KUKA KRL program: test1.src, test1.dat

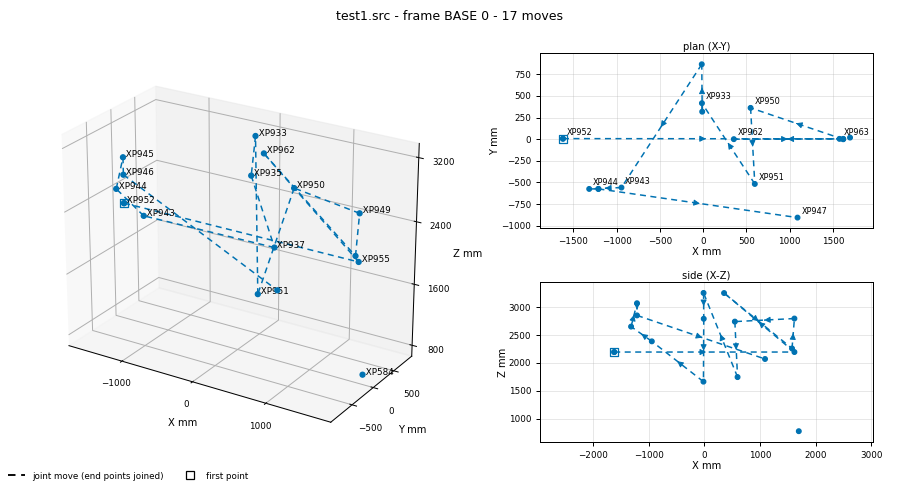
[picture p0: tool path of test1.src in frame BASE 0, 17 of 19 moves have a stored position in this frame; points joined in program order, loops and branches not executed]
--- test1.src ---
&ACCESS RVP
&REL 764
&PARAM TEMPLATE = C:\KRC\Roboter\Template\vorgabe
&PARAM EDITMASK = *
DEF test1( )
;FOLD INI;%{PE}%V3.2.0,%MKUKATPBASIS,%CINIT,%VCOMMON,%P
;FOLD BAS INI;%{E}%V3.2.0,%MKUKATPBASIS,%CINIT,%VINIT,%P
GLOBAL INTERRUPT DECL 3 WHEN $STOPMESS==TRUE DO IR_STOPM ( )
INTERRUPT ON 3
BAS (#INITMOV,0 )
;ENDFOLD (BAS INI)
;FOLD A20 INI;%{E}%V3.2.0,%MKUKATPA20,%CINIT,%VINIT,%P
IF ARC20==TRUE THEN
A20 (ARC_INI)
INTERRUPT DECL 6 WHEN $CYCFLAG[3]==FALSE DO A20(TECH_STOP2)
ENDIF
;ENDFOLD (A20 INI)
;FOLD A10 INI;%{E}%V3.2.0,%MKUKATPARC,%CINIT,%VINIT,%P
IF A10_OPTION==#ACTIVE THEN
INTERRUPT DECL 4 WHEN $CYCFLAG[2]==FALSE DO A10 (#APPL_ERROR)
INTERRUPT DECL 7 WHEN A_ARC_SWI==#ACTIVE DO A10 (#ARC_SEAM)
INTERRUPT DECL 5 WHEN A_FLY_ARC==TRUE DO A10 (#HPU_ARC)
INTERRUPT  ON 5
A10_INI ( )
ENDIF
;ENDFOLD (A10 INI)
;FOLD GRIPPER INI;%{E}%V3.2.0,%MKUKATPGRIPPER,%CINIT,%VINIT,%P
USER_GRP(0,DUMMY,DUMMY,GDEFAULT)
;ENDFOLD (GRIPPER INI)
;FOLD SPOT INI;%{E}%V3.2.0,%MKUKATPSPOT,%CINIT,%VINIT,%P
USERSPOT(#INIT)
;ENDFOLD (SPOT INI)
;FOLD TOUCHSENSE INI;%{E}%V3.2.0,%MKUKATPTS,%CINIT,%VINIT,%P
IF H70_OPTION THEN
INTERRUPT DECL 15 WHEN $MEAS_PULSE[TOUCH_I[TOUCH_ACTIVE].IN_NR] DO H70 (6,CD0 )
INTERRUPT DECL 16 WHEN $ZERO_MOVE DO H70 (7,CD0 )
INTERRUPT DECL 17 WHEN $TECHPAR_C[FG_TOUCH,8]>0.5 DO H70 (8,CD0)
H70 (1,CD0 )
ENDIF
;ENDFOLD (TOUCHSENSE INI)
;FOLD USER INI;%{E}%V3.2.0,%MKUKATPUSER,%CINIT,%VINIT,%P
;Make your modifications here
;ENDFOLD (USER INI)
;ENDFOLD (INI)
loop
;FOLD PTP HOME  Vel= 100 % DEFAULT;%{PE}%R 4.1.16,%MKUKATPBASIS,%CMOVE,%VPTP,%P 1:PTP, 2:HOME, 3:, 5:100, 7:DEFAULT
$BWDSTART = FALSE
PDAT_ACT=PDEFAULT
BAS(#PTP_DAT)
FDAT_ACT=FHOME
BAS(#FRAMES)
BAS(#VEL_PTP,100)
$H_POS=XHOME
PTP XHOME
;ENDFOLD


;FOLD WAIT Time= 2 sec;%{PE}%R 4.1.16,%MKUKATPBASIS,%CWAIT,%VWAIT,%P 2:2
WAIT SEC 2
;ENDFOLD

;FOLD PTP P952  Vel= 50 % PDAT628 Tool[1] Base[0];%{PE}%R 4.1.16,%MKUKATPBASIS,%CMOVE,%VPTP,%P 1:PTP, 2:P952, 3:, 5:50, 7:PDAT628
$BWDSTART = FALSE
PDAT_ACT=PPDAT628
BAS(#PTP_DAT)
FDAT_ACT=FP952
BAS(#FRAMES)
BAS(#VEL_PTP,50)
PTP XP952
;ENDFOLD
;FOLD PTP P954  Vel= 50 % PDAT630 Tool[1] Base[0];%{PE}%R 4.1.16,%MKUKATPBASIS,%CMOVE,%VPTP,%P 1:PTP, 2:P954, 3:, 5:50, 7:PDAT630
$BWDSTART = FALSE
PDAT_ACT=PPDAT630
BAS(#PTP_DAT)
FDAT_ACT=FP954
BAS(#FRAMES)
BAS(#VEL_PTP,50)
PTP XP954
;ENDFOLD
;FOLD PTP P955 CONT Vel= 100 % PDAT631 Tool[1]:Lexan Pointer Base[0];%{PE}%R 4.1.16,%MKUKATPBASIS,%CMOVE,%VPTP,%P 1:PTP, 2:P955, 3:C_PTP, 5:100, 7:PDAT631
$BWDSTART = FALSE
PDAT_ACT=PPDAT631
BAS(#PTP_DAT)
FDAT_ACT=FP955
BAS(#FRAMES)
BAS(#VEL_PTP,100)
PTP XP955 C_PTP
;ENDFOLD
;FOLD PTP P962 CONT Vel= 100 % PDAT638 Tool[1]:Lexan Pointer Base[0];%{PE}%R 4.1.16,%MKUKATPBASIS,%CMOVE,%VPTP,%P 1:PTP, 2:P962, 3:C_PTP, 5:100, 7:PDAT638
$BWDSTART = FALSE
PDAT_ACT=PPDAT638
BAS(#PTP_DAT)
FDAT_ACT=FP962
BAS(#FRAMES)
BAS(#VEL_PTP,100)
PTP XP962 C_PTP
;ENDFOLD
;FOLD PTP P963 CONT Vel= 100 % PDAT639 Tool[1]:Lexan Pointer Base[0];%{PE}%R 4.1.16,%MKUKATPBASIS,%CMOVE,%VPTP,%P 1:PTP, 2:P963, 3:C_PTP, 5:100, 7:PDAT639
$BWDSTART = FALSE
PDAT_ACT=PPDAT639
BAS(#PTP_DAT)
FDAT_ACT=FP963
BAS(#FRAMES)
BAS(#VEL_PTP,100)
PTP XP963 C_PTP
;ENDFOLD
;FOLD PTP P949 CONT Vel= 100 % PDAT625 Tool[1]:Lexan Pointer Base[0];%{PE}%R 4.1.16,%MKUKATPBASIS,%CMOVE,%VPTP,%P 1:PTP, 2:P949, 3:C_PTP, 5:100, 7:PDAT625
$BWDSTART = FALSE
PDAT_ACT=PPDAT625
BAS(#PTP_DAT)
FDAT_ACT=FP949
BAS(#FRAMES)
BAS(#VEL_PTP,100)
PTP XP949 C_PTP
;ENDFOLD

;FOLD PTP P950 CONT Vel= 100 % PDAT626 Tool[1]:Lexan Pointer Base[0];%{PE}%R 4.1.16,%MKUKATPBASIS,%CMOVE,%VPTP,%P 1:PTP, 2:P950, 3:C_PTP, 5:100, 7:PDAT626
$BWDSTART = FALSE
PDAT_ACT=PPDAT626
BAS(#PTP_DAT)
FDAT_ACT=FP950
BAS(#FRAMES)
BAS(#VEL_PTP,100)
PTP XP950 C_PTP
;ENDFOLD
;FOLD PTP P951 CONT Vel= 100 % PDAT627 Tool[1]:Lexan Pointer Base[0];%{PE}%R 4.1.16,%MKUKATPBASIS,%CMOVE,%VPTP,%P 1:PTP, 2:P951, 3:C_PTP, 5:100, 7:PDAT627
$BWDSTART = FALSE
PDAT_ACT=PPDAT627
BAS(#PTP_DAT)
FDAT_ACT=FP951
BAS(#FRAMES)
BAS(#VEL_PTP,100)
PTP XP951 C_PTP
;ENDFOLD
;FOLD PTP P933 CONT Vel= 100 % PDAT609 Tool[1]:Lexan Pointer Base[0];%{PE}%R 4.1.16,%MKUKATPBASIS,%CMOVE,%VPTP,%P 1:PTP, 2:P933, 3:C_PTP, 5:100, 7:PDAT609
$BWDSTART = FALSE
PDAT_ACT=PPDAT609
BAS(#PTP_DAT)
FDAT_ACT=FP933
BAS(#FRAMES)
BAS(#VEL_PTP,100)
PTP XP933 C_PTP
;ENDFOLD
;FOLD PTP P935 CONT Vel= 100 % PDAT611 Tool[1]:Lexan Pointer Base[0];%{PE}%R 4.1.16,%MKUKATPBASIS,%CMOVE,%VPTP,%P 1:PTP, 2:P935, 3:C_PTP, 5:100, 7:PDAT611
$BWDSTART = FALSE
PDAT_ACT=PPDAT611
BAS(#PTP_DAT)
FDAT_ACT=FP935
BAS(#FRAMES)
BAS(#VEL_PTP,100)
PTP XP935 C_PTP
;ENDFOLD
;FOLD PTP P937 CONT Vel= 100 % PDAT613 Tool[1]:Lexan Pointer Base[0];%{PE}%R 4.1.16,%MKUKATPBASIS,%CMOVE,%VPTP,%P 1:PTP, 2:P937, 3:C_PTP, 5:100, 7:PDAT613
$BWDSTART = FALSE
PDAT_ACT=PPDAT613
BAS(#PTP_DAT)
FDAT_ACT=FP937
BAS(#FRAMES)
BAS(#VEL_PTP,100)
PTP XP937 C_PTP
;ENDFOLD



;FOLD ; Robot is now at ship;%{PE}%R 4.1.16,%MKUKATPBASIS,%CCOMMENT,%VNORMAL,%P 2:Robot is now at ship
;ENDFOLD

;FOLD PTP P943 CONT Vel= 100 % PDAT619 Tool[1]:Lexan Pointer Base[0];%{PE}%R 4.1.16,%MKUKATPBASIS,%CMOVE,%VPTP,%P 1:PTP, 2:P943, 3:C_PTP, 5:100, 7:PDAT619
$BWDSTART = FALSE
PDAT_ACT=PPDAT619
BAS(#PTP_DAT)
FDAT_ACT=FP943
BAS(#FRAMES)
BAS(#VEL_PTP,100)
PTP XP943 C_PTP
;ENDFOLD
;FOLD PTP P944 CONT Vel= 100 % PDAT620 Tool[1]:Lexan Pointer Base[0];%{PE}%R 4.1.16,%MKUKATPBASIS,%CMOVE,%VPTP,%P 1:PTP, 2:P944, 3:C_PTP, 5:100, 7:PDAT620
$BWDSTART = FALSE
PDAT_ACT=PPDAT620
BAS(#PTP_DAT)
FDAT_ACT=FP944
BAS(#FRAMES)
BAS(#VEL_PTP,100)
PTP XP944 C_PTP
;ENDFOLD
;FOLD PTP P945 CONT Vel= 100 % PDAT621 Tool[1]:Lexan Pointer Base[0];%{PE}%R 4.1.16,%MKUKATPBASIS,%CMOVE,%VPTP,%P 1:PTP, 2:P945, 3:C_PTP, 5:100, 7:PDAT621
$BWDSTART = FALSE
PDAT_ACT=PPDAT621
BAS(#PTP_DAT)
FDAT_ACT=FP945
BAS(#FRAMES)
BAS(#VEL_PTP,100)
PTP XP945 C_PTP
;ENDFOLD
;FOLD PTP P946 CONT Vel= 100 % PDAT622 Tool[1]:Lexan Pointer Base[0];%{PE}%R 4.1.16,%MKUKATPBASIS,%CMOVE,%VPTP,%P 1:PTP, 2:P946, 3:C_PTP, 5:100, 7:PDAT622
$BWDSTART = FALSE
PDAT_ACT=PPDAT622
BAS(#PTP_DAT)
FDAT_ACT=FP946
BAS(#FRAMES)
BAS(#VEL_PTP,100)
PTP XP946 C_PTP
;ENDFOLD
;FOLD PTP P947 CONT Vel= 100 % PDAT623 Tool[1]:Lexan Pointer Base[0];%{PE}%R 4.1.16,%MKUKATPBASIS,%CMOVE,%VPTP,%P 1:PTP, 2:P947, 3:C_PTP, 5:100, 7:PDAT623
$BWDSTART = FALSE
PDAT_ACT=PPDAT623
BAS(#PTP_DAT)
FDAT_ACT=FP947
BAS(#FRAMES)
BAS(#VEL_PTP,100)
PTP XP947 C_PTP
;ENDFOLD

;FOLD ; Begin with tower 1;%{PE}%R 4.1.16,%MKUKATPBASIS,%CCOMMENT,%VNORMAL,%P 2:Begin with tower 1
;ENDFOLD


;FOLD ; tower 2 done;%{PE}%R 4.1.16,%MKUKATPBASIS,%CCOMMENT,%VNORMAL,%P 2:tower 2 done
;ENDFOLD
;FOLD ; approach;%{PE}%R 4.1.16,%MKUKATPBASIS,%CCOMMENT,%VNORMAL,%P 2:approach
;ENDFOLD



;FOLD ; foreword approach;%{PE}%R 4.1.16,%MKUKATPBASIS,%CCOMMENT,%VNORMAL,%P 2:foreword approach
;ENDFOLD







;FOLD ; mouth;%{PE}%R 4.1.16,%MKUKATPBASIS,%CCOMMENT,%VNORMAL,%P 2:mouth
;ENDFOLD

;FOLD ; top vert orbit;%{PE}%R 4.1.16,%MKUKATPBASIS,%CCOMMENT,%VNORMAL,%P 2:top vert orbit
;ENDFOLD



;FOLD ; mid orbit;%{PE}%R 4.1.16,%MKUKATPBASIS,%CCOMMENT,%VNORMAL,%P 2:mid orbit
;ENDFOLD














;FOLD PTP HOME CONT Vel= 50 % DEFAULT;%{PE}%R 4.1.16,%MKUKATPBASIS,%CMOVE,%VPTP,%P 1:PTP, 2:HOME, 3:C_PTP, 5:50, 7:DEFAULT
$BWDSTART = FALSE
PDAT_ACT=PDEFAULT
BAS(#PTP_DAT)
FDAT_ACT=FHOME
BAS(#FRAMES)
BAS(#VEL_PTP,50)
$H_POS=XHOME
PTP XHOME C_PTP
;ENDFOLD
endloop


;FOLD ; paul center index1;%{PE}%R 4.1.16,%MKUKATPBASIS,%CCOMMENT,%VNORMAL,%P 2:paul center index1
;ENDFOLD
;FOLD PTP P584  Vel= 100 % PDAT377 Tool[1]:Lexan Pointer Base[0];%{PE}%R 4.1.16,%MKUKATPBASIS,%CMOVE,%VPTP,%P 1:PTP, 2:P584, 3:, 5:100, 7:PDAT377
$BWDSTART = FALSE
PDAT_ACT=PPDAT377
BAS(#PTP_DAT)
FDAT_ACT=FP584
BAS(#FRAMES)
BAS(#VEL_PTP,100)
PTP XP584
;ENDFOLD


END

--- test1.dat ---
&ACCESS RVP
&REL 764
&PARAM TEMPLATE = C:\KRC\Roboter\Template\vorgabe
&PARAM EDITMASK = *
DEFDAT  TEST1
;FOLD EXTERNAL DECLARATIONS;%{PE}%V3.2.0,%MKUKATPBASIS,%CEXT,%VCOMMON,%P
;FOLD BAS EXT;%{PE}%V3.2.0,%MKUKATPBASIS,%CEXT,%VEXT,%P
EXT  BAS (BAS_COMMAND  :IN,REAL  :IN )
DECL INT SUCCESS
;ENDFOLD
;FOLD A10 EXT;%{E}%V3.2.0,%MKUKATPARC,%CEXT,%VEXT,%P
EXT  A10 (A_CMD_T  :IN,A_STRT_T  :IN,A_WELD_T  :IN,A_END_T  :IN,INT  :IN )
;ENDFOLD
;FOLD A20 EXT;%{E}%V3.2.0,%MKUKATPA20,%CEXT,%VEXT,%P
EXT  A20 (INT  :IN,WELD_ST  :IN,WELD_FI  :IN,INT  :IN )
;ENDFOLD
;FOLD GRIPPER EXT;%{E}%V3.2.0,%MKUKATPGRIPPER,%CEXT,%VEXT,%P
EXT  H50 (INT  :IN,INT  :IN,INT  :IN,GRP_TYP  :IN )
;ENDFOLD
;FOLD SPOT EXT;%{E}%V3.2.0,%MKUKATPSPOT,%CEXT,%VEXT,%P
EXT  USERSPOT (S_COMMAND  :IN,SPOT_TYPE  :IN )
;ENDFOLD
;FOLD TOUCHSENSE EXT;%{E}%V3.2.0,%MKUKATPTS,%CEXT,%VEXT,%P
EXT  H70 (INT  :IN,SRCH_TYP_2  :OUT,E6POS  :IN,SRCH_TYP_3  :IN,SRCH_TYP_2  :IN,SRCH_TYP_2  :IN,SRCH_TYP_2  :IN,SRCH_TYP_2  :IN,SRCH_TYP_2  :IN,INT  :IN )
;ENDFOLD
;FOLD USER EXT;%{E}%V3.2.0,%MKUKATPUSER,%CEXT,%VEXT,%P
;Make here your modifications
;ENDFOLD
;ENDFOLD

DECL E6POS XP1={x 22.64711,y 0.635935128,z 3052.04297,a 80.9998016,b 0.750907719,c 2.94084597,s 6,t 50,e1 0.0,e2 0.0,e3 0.0,e4 0.0,e5 0.0,e6 0.0}
DECL BASIS_SUGG_T LAST_BASIS={POINT1[] "P974                    ",POINT2[] "P974                    ",CP_PARAMS[] "CPDAT294                ",PTP_PARAMS[] "PDAT650                 ",CONT[] "C_PTP                   ",CP_VEL[] "0.1                     ",PTP_VEL[] "100                     "}
DECL FDAT FP1={TOOL_NO 1,BASE_NO 0,IPO_FRAME #BASE}
DECL PDAT PPDAT1={VEL 100.0,ACC 100.0,APO_DIST 100.0}
DECL E6POS XP2={x -317.379913,y 28.4180508,z 3098.27002,a 81.0803528,b -1.12059498,c -21.6292801,s 7,t 50,e1 0.0,e2 0.0,e3 0.0,e4 0.0,e5 0.0,e6 0.0}
DECL FDAT FP2={TOOL_NO 1,BASE_NO 0,IPO_FRAME #BASE}
DECL PDAT PPDAT2={VEL 100.0,ACC 100.0,APO_DIST 100.0}
DECL E6POS XP3={x -1118.88,y 93.9099884,z 2113.15601,a 84.8656082,b -4.36905909,c -90.8236465,s 5,t 54,e1 0.0,e2 0.0,e3 0.0,e4 0.0,e5 0.0,e6 0.0}
DECL FDAT FP3={TOOL_NO 1,BASE_NO 0,IPO_FRAME #BASE}
DECL PDAT PPDAT3={VEL 100.0,ACC 100.0,APO_DIST 100.0}
DECL E6POS XP4={x -914.403687,y 77.2060089,z 1371.20605,a 87.7985306,b -3.63463497,c -131.1138,s 5,t 54,e1 0.0,e2 0.0,e3 0.0,e4 0.0,e5 0.0,e6 0.0}
DECL FDAT FP4={TOOL_NO 1,BASE_NO 0,IPO_FRAME #BASE}
DECL PDAT PPDAT4={VEL 100.0,ACC 100.0,APO_DIST 100.0}
DECL E6POS XP5={x 456.821198,y 795.871826,z 1371.20801,a -27.2306709,b -3.63450098,c -131.113693,s 5,t 54,e1 0.0,e2 0.0,e3 0.0,e4 0.0,e5 0.0,e6 0.0}
DECL FDAT FP5={TOOL_NO 1,BASE_NO 0,IPO_FRAME #BASE}
DECL PDAT PPDAT5={VEL 100.0,ACC 100.0,APO_DIST 100.0}
DECL E6POS XP6={x 279.509613,y 463.9599,z 1341.03894,a 63.2674294,b 39.8199005,c 179.158493,s 5,t 22,e1 0.0,e2 0.0,e3 0.0,e4 0.0,e5 0.0,e6 0.0}
DECL FDAT FP6={TOOL_NO 1,BASE_NO 0,IPO_FRAME #BASE}
DECL PDAT PPDAT6={VEL 100.0,ACC 100.0,APO_DIST 100.0}
DECL E6POS XP7={x 342.425201,y 611.915222,z 1278.76099,a -117.584503,b -2.66220593,c 178.681595,s 1,t 14,e1 0.0,e2 0.0,e3 0.0,e4 0.0,e5 0.0,e6 0.0}
DECL FDAT FP7={TOOL_NO 1,BASE_NO 0,IPO_FRAME #BASE}
DECL PDAT PPDAT7={VEL 100.0,ACC 100.0,APO_DIST 100.0}
DECL E6POS XP8={x -383.700897,y 898.310181,z 2029.78894,a -64.2966537,b 43.4239197,c -179.217896,s 1,t 14,e1 0.0,e2 0.0,e3 0.0,e4 0.0,e5 0.0,e6 0.0}
DECL FDAT FP8={TOOL_NO 1,BASE_NO 0,IPO_FRAME #BASE}
DECL PDAT PPDAT8={VEL 100.0,ACC 100.0,APO_DIST 100.0}
DECL E6POS XP9={x -686.96521,y 252.598007,z 2706.76709,a 1.83803499,b 84.4630966,c -158.838196,s 1,t 14,e1 0.0,e2 0.0,e3 0.0,e4 0.0,e5 0.0,e6 0.0}
DECL FDAT FP9={TOOL_NO 1,BASE_NO 0,IPO_FRAME #BASE}
DECL PDAT PPDAT9={VEL 100.0,ACC 100.0,APO_DIST 100.0}
DECL E6POS XP10={x -287.330109,y 102.080002,z 2968.2041,a 155.448105,b 57.2829208,c -4.51428509,s 3,t 10,e1 0.0,e2 0.0,e3 0.0,e4 0.0,e5 0.0,e6 0.0}
DECL FDAT FP10={TOOL_NO 1,BASE_NO 0,IPO_FRAME #BASE}
DECL PDAT PPDAT10={VEL 100.0,ACC 100.0,APO_DIST 100.0}
DECL E6POS XP11={x 756.905884,y -474.43161,z 2068.03589,a -175.991699,b 26.8178406,c -123.306099,s 2,t 10,e1 0.0,e2 0.0,e3 0.0,e4 0.0,e5 0.0,e6 0.0}
DECL FDAT FP11={TOOL_NO 1,BASE_NO 0,IPO_FRAME #BASE}
DECL PDAT PPDAT11={VEL 100.0,ACC 100.0,APO_DIST 100.0}
DECL E6POS XP12={x 737.561218,y -322.266388,z 1746.229,a 167.528503,b 26.5866203,c -167.384705,s 2,t 10,e1 0.0,e2 0.0,e3 0.0,e4 0.0,e5 0.0,e6 0.0}
DECL FDAT FP12={TOOL_NO 1,BASE_NO 0,IPO_FRAME #BASE}
DECL PDAT PPDAT12={VEL 100.0,ACC 100.0,APO_DIST 100.0}
DECL E6POS XP13={x 727.209717,y -62.4198189,z 1656.07202,a 86.3765564,b -0.340090901,c 166.081207,s 2,t 42,e1 0.0,e2 0.0,e3 0.0,e4 0.0,e5 0.0,e6 0.0}
DECL FDAT FP13={TOOL_NO 1,BASE_NO 0,IPO_FRAME #BASE}
DECL PDAT PPDAT13={VEL 100.0,ACC 100.0,APO_DIST 100.0}
DECL E6POS XP14={x 930.632996,y -86.8171768,z 1931.13501,a -95.5554962,b 3.7291801,c -87.2372894,s 2,t 34,e1 0.0,e2 0.0,e3 0.0,e4 0.0,e5 0.0,e6 0.0}
DECL FDAT FP14={TOOL_NO 1,BASE_NO 0,IPO_FRAME #BASE}
DECL PDAT PPDAT14={VEL 100.0,ACC 100.0,APO_DIST 100.0}
DECL E6POS XP15={x 877.973511,y -96.1897888,z 1759.84399,a 86.188652,b 7.87783909,c 126.2939,s 2,t 34,e1 0.0,e2 0.0,e3 0.0,e4 0.0,e5 0.0,e6 0.0}
DECL FDAT FP15={TOOL_NO 1,BASE_NO 0,IPO_FRAME #BASE}
DECL PDAT PPDAT15={VEL 100.0,ACC 100.0,APO_DIST 100.0}
DECL E6POS XP16={x 854.0224,y -94.0261002,z 2184.73608,a 83.0226517,b 7.78562021,c 103.365303,s 2,t 34,e1 0.0,e2 0.0,e3 0.0,e4 0.0,e5 0.0,e6 0.0}
DECL FDAT FP16={TOOL_NO 1,BASE_NO 0,IPO_FRAME #BASE}
DECL PDAT PPDAT16={VEL 100.0,ACC 100.0,APO_DIST 100.0}
DECL E6POS XP17={x 859.931885,y -94.021843,z 1948.71997,a 84.9119034,b 6.17852592,c 123.187599,s 2,t 34,e1 0.0,e2 0.0,e3 0.0,e4 0.0,e5 0.0,e6 0.0}
DECL FDAT FP17={TOOL_NO 1,BASE_NO 0,IPO_FRAME #BASE}
DECL PDAT PPDAT17={VEL 100.0,ACC 100.0,APO_DIST 100.0}
DECL E6POS XP18={x 859.932312,y -30.10009,z 2284.0271,a 84.9120865,b 6.17841005,c 123.187698,s 2,t 35,e1 0.0,e2 0.0,e3 0.0,e4 0.0,e5 0.0,e6 0.0}
DECL FDAT FP18={TOOL_NO 1,BASE_NO 0,IPO_FRAME #BASE}
DECL PDAT PPDAT18={VEL 100.0,ACC 100.0,APO_DIST 100.0}
DECL E6POS XP19={x 860.002197,y -30.1490498,z 2284.14795,a 82.0233612,b 0.703113616,c 77.8308716,s 2,t 35,e1 0.0,e2 0.0,e3 0.0,e4 0.0,e5 0.0,e6 0.0}
DECL FDAT FP19={TOOL_NO 1,BASE_NO 0,IPO_FRAME #BASE}
DECL PDAT PPDAT19={VEL 100.0,ACC 100.0,APO_DIST 100.0}
DECL E6POS XP20={x 860.007874,y -30.1515293,z 2284.1521,a -75.3501968,b -56.7245789,c -114.399101,s 2,t 34,e1 0.0,e2 0.0,e3 0.0,e4 0.0,e5 0.0,e6 0.0}
DECL FDAT FP20={TOOL_NO 1,BASE_NO 0,IPO_FRAME #BASE}
DECL PDAT PPDAT20={VEL 100.0,ACC 100.0,APO_DIST 100.0}
DECL E6POS XP21={x 860.005188,y -30.1509609,z 2284.16089,a 76.9720535,b -27.3394794,c 104.781601,s 2,t 34,e1 0.0,e2 0.0,e3 0.0,e4 0.0,e5 0.0,e6 0.0}
DECL FDAT FP21={TOOL_NO 1,BASE_NO 0,IPO_FRAME #BASE}
DECL PDAT PPDAT21={VEL 100.0,ACC 100.0,APO_DIST 100.0}
DECL E6POS XP22={x 902.046509,y -30.2999706,z 1758.10901,a 65.3865967,b -17.9801807,c 134.1922,s 2,t 34,e1 0.0,e2 0.0,e3 0.0,e4 0.0,e5 0.0,e6 0.0}
DECL FDAT FP22={TOOL_NO 1,BASE_NO 0,IPO_FRAME #BASE}
DECL PDAT PPDAT22={VEL 100.0,ACC 100.0,APO_DIST 100.0}
DECL E6POS XP23={x -2.01831698,y -399.759613,z 2936.4939,a 25.6383991,b -0.42615509,c 10.0116596,s 6,t 50,e1 0.0,e2 0.0,e3 0.0,e4 0.0,e5 0.0,e6 0.0}
DECL FDAT FP23={TOOL_NO 1,BASE_NO 0,IPO_FRAME #BASE}
DECL PDAT PPDAT23={VEL 100.0,ACC 100.0,APO_DIST 100.0}
DECL E6POS XP24={x 366.294403,y -40.3560295,z 2954.28711,a 106.809502,b -13.3838701,c 28.0512791,s 2,t 34,e1 0.0,e2 0.0,e3 0.0,e4 0.0,e5 0.0,e6 0.0}
DECL FDAT FP24={TOOL_NO 1,BASE_NO 0,IPO_FRAME #BASE}
DECL PDAT PPDAT24={VEL 100.0,ACC 100.0,APO_DIST 100.0}
DECL E6POS XP25={x -96.3233337,y -16.0035496,z 3109.52197,a 124.831001,b -1.57262802,c 2.47217989,s 3,t 35,e1 0.0,e2 0.0,e3 0.0,e4 0.0,e5 0.0,e6 0.0}
DECL FDAT FP25={TOOL_NO 1,BASE_NO 0,IPO_FRAME #BASE}
DECL PDAT PPDAT25={VEL 100.0,ACC 100.0,APO_DIST 100.0}
DECL E6POS XP26={x -265.2453,y -105.245903,z 3116.50391,a 137.165894,b 5.24283218,c -11.4044304,s 3,t 35,e1 0.0,e2 0.0,e3 0.0,e4 0.0,e5 0.0,e6 0.0}
DECL FDAT FP26={TOOL_NO 1,BASE_NO 0,IPO_FRAME #BASE}
DECL PDAT PPDAT26={VEL 100.0,ACC 100.0,APO_DIST 100.0}
DECL E6POS XP27={x -382.447388,y 15.0625801,z 2903.76099,a 169.007996,b -1.03763604,c 42.8505402,s 1,t 47,e1 0.0,e2 0.0,e3 0.0,e4 0.0,e5 0.0,e6 0.0}
DECL FDAT FP27={TOOL_NO 1,BASE_NO 0,IPO_FRAME #BASE}
DECL PDAT PPDAT27={VEL 100.0,ACC 100.0,APO_DIST 100.0}
DECL E6POS XP28={x 314.934998,y 163.138,z 2876.17603,a 134.743607,b -43.0532684,c 78.4436188,s 2,t 43,e1 0.0,e2 0.0,e3 0.0,e4 0.0,e5 0.0,e6 0.0}
DECL FDAT FP28={TOOL_NO 1,BASE_NO 0,IPO_FRAME #BASE}
DECL PDAT PPDAT28={VEL 100.0,ACC 100.0,APO_DIST 100.0}
DECL E6POS XP29={x 874.750488,y 15.4131098,z 2242.91992,a -54.1314201,b 11.3628597,c -11.9078903,s 2,t 43,e1 0.0,e2 0.0,e3 0.0,e4 0.0,e5 0.0,e6 0.0}
DECL FDAT FP29={TOOL_NO 1,BASE_NO 0,IPO_FRAME #BASE}
DECL PDAT PPDAT29={VEL 100.0,ACC 100.0,APO_DIST 100.0}
DECL E6POS XP30={x 763.66803,y 12.42836,z 2062.2981,a -53.9077797,b 0.727466524,c 3.2328341,s 2,t 43,e1 0.0,e2 0.0,e3 0.0,e4 0.0,e5 0.0,e6 0.0}
DECL FDAT FP30={TOOL_NO 1,BASE_NO 0,IPO_FRAME #BASE}
DECL PDAT PPDAT30={VEL 100.0,ACC 100.0,APO_DIST 100.0}
DECL E6POS XP31={x 627.086914,y -123.824997,z 1621.20605,a 61.813221,b 49.352169,c -167.257904,s 2,t 43,e1 0.0,e2 0.0,e3 0.0,e4 0.0,e5 0.0,e6 0.0}
DECL FDAT FP31={TOOL_NO 1,BASE_NO 0,IPO_FRAME #BASE}
DECL PDAT PPDAT31={VEL 100.0,ACC 100.0,APO_DIST 100.0}
DECL E6POS XP32={x 872.744019,y 4.39807701,z 1542.26001,a -119.030197,b 6.9775281,c -159.180603,s 6,t 59,e1 0.0,e2 0.0,e3 0.0,e4 0.0,e5 0.0,e6 0.0}
DECL FDAT FP32={TOOL_NO 1,BASE_NO 0,IPO_FRAME #BASE}
DECL PDAT PPDAT32={VEL 100.0,ACC 100.0,APO_DIST 100.0}
DECL E6POS XP33={x 987.663818,y 54.8688316,z 1954.90503,a -64.3430328,b 21.8002701,c -49.7024918,s 2,t 43,e1 0.0,e2 0.0,e3 0.0,e4 0.0,e5 0.0,e6 0.0}
DECL FDAT FP33={TOOL_NO 1,BASE_NO 0,IPO_FRAME #BASE}
DECL PDAT PPDAT33={VEL 100.0,ACC 100.0,APO_DIST 100.0}
DECL E6POS XP34={x 987.665283,y 54.8672905,z 1954.91394,a 142.235794,b -42.7988892,c 35.0734596,s 2,t 43,e1 0.0,e2 0.0,e3 0.0,e4 0.0,e5 0.0,e6 0.0}
DECL FDAT FP34={TOOL_NO 1,BASE_NO 0,IPO_FRAME #BASE}
DECL PDAT PPDAT34={VEL 100.0,ACC 100.0,APO_DIST 100.0}
DECL E6POS XP35={x 848.862976,y -115.089996,z 1573.91895,a -108.386902,b -26.3736305,c -154.792404,s 2,t 43,e1 0.0,e2 0.0,e3 0.0,e4 0.0,e5 0.0,e6 0.0}
DECL FDAT FP35={TOOL_NO 1,BASE_NO 0,IPO_FRAME #BASE}
DECL PDAT PPDAT35={VEL 100.0,ACC 100.0,APO_DIST 100.0}
DECL E6POS XP36={x 919.167114,y -112.897903,z 2081.95996,a -115.377701,b -19.0544605,c -136.852097,s 2,t 43,e1 0.0,e2 0.0,e3 0.0,e4 0.0,e5 0.0,e6 0.0}
DECL FDAT FP36={TOOL_NO 1,BASE_NO 0,IPO_FRAME #BASE}
DECL PDAT PPDAT36={VEL 100.0,ACC 100.0,APO_DIST 100.0}
DECL E6POS XP37={x 919.275696,y -112.841904,z 2081.85693,a -121.187599,b 3.30841398,c -96.9181213,s 2,t 43,e1 0.0,e2 0.0,e3 0.0,e4 0.0,e5 0.0,e6 0.0}
DECL FDAT FP37={TOOL_NO 1,BASE_NO 0,IPO_FRAME #BASE}
DECL PDAT PPDAT37={VEL 100.0,ACC 100.0,APO_DIST 100.0}
DECL E6POS XP38={x 911.011902,y -133.252304,z 2112.41406,a -119.583099,b -23.0007591,c -108.861801,s 2,t 43,e1 0.0,e2 0.0,e3 0.0,e4 0.0,e5 0.0,e6 0.0}
DECL FDAT FP38={TOOL_NO 1,BASE_NO 0,IPO_FRAME #BASE}
DECL PDAT PPDAT38={VEL 100.0,ACC 100.0,APO_DIST 100.0}
DECL E6POS XP39={x 699.043884,y 284.058807,z 2125.91089,a 36.3473206,b -65.9336319,c -127.379204,s 6,t 59,e1 0.0,e2 0.0,e3 0.0,e4 0.0,e5 0.0,e6 0.0}
DECL FDAT FP39={TOOL_NO 1,BASE_NO 0,IPO_FRAME #BASE}
DECL PDAT PPDAT39={VEL 100.0,ACC 100.0,APO_DIST 100.0}
DECL E6POS XP40={x 934.429504,y -100.2621,z 2266.78809,a -146.033203,b -58.5612297,c -58.2801895,s 2,t 43,e1 0.0,e2 0.0,e3 0.0,e4 0.0,e5 0.0,e6 0.0}
DECL FDAT FP40={TOOL_NO 1,BASE_NO 0,IPO_FRAME #BASE}
DECL PDAT PPDAT40={VEL 100.0,ACC 100.0,APO_DIST 100.0}
DECL E6POS XP41={x 704.38623,y -242.486404,z 2244.26196,a 168.325607,b -45.4726791,c -74.2092972,s 2,t 43,e1 0.0,e2 0.0,e3 0.0,e4 0.0,e5 0.0,e6 0.0}
DECL FDAT FP41={TOOL_NO 1,BASE_NO 0,IPO_FRAME #BASE}
DECL PDAT PPDAT41={VEL 100.0,ACC 100.0,APO_DIST 100.0}
DECL E6POS XP42={x 753.340088,y 29.5257893,z 2458.37305,a 122.371803,b -4.2261591,c 9.3760004,s 2,t 43,e1 0.0,e2 0.0,e3 0.0,e4 0.0,e5 0.0,e6 0.0}
DECL FDAT FP42={TOOL_NO 1,BASE_NO 0,IPO_FRAME #BASE}
DECL PDAT PPDAT42={VEL 100.0,ACC 100.0,APO_DIST 100.0}
DECL E6POS XP43={x 752.161682,y 18.1640797,z 1926.76404,a 60.7446518,b -4.06174803,c 170.900299,s 6,t 59,e1 0.0,e2 0.0,e3 0.0,e4 0.0,e5 0.0,e6 0.0}
DECL FDAT FP43={TOOL_NO 1,BASE_NO 0,IPO_FRAME #BASE}
DECL PDAT PPDAT43={VEL 100.0,ACC 100.0,APO_DIST 100.0}
DECL E6POS XP44={x 963.605286,y 37.0490417,z 2271.19702,a 81.6219635,b 33.4775085,c 69.5978088,s 6,t 59,e1 0.0,e2 0.0,e3 0.0,e4 0.0,e5 0.0,e6 0.0}
DECL FDAT FP44={TOOL_NO 1,BASE_NO 0,IPO_FRAME #BASE}
DECL PDAT PPDAT44={VEL 100.0,ACC 100.0,APO_DIST 100.0}
DECL E6POS XP45={x 959.966125,y 42.6314507,z 2289.33691,a 83.5021973,b 33.1825409,c 72.5745697,s 6,t 59,e1 0.0,e2 0.0,e3 0.0,e4 0.0,e5 0.0,e6 0.0}
DECL FDAT FP45={TOOL_NO 1,BASE_NO 0,IPO_FRAME #BASE}
DECL PDAT PPDAT45={VEL 100.0,ACC 100.0,APO_DIST 100.0}
DECL E6POS XP46={x 959.931519,y 42.6475487,z 2285.76611,a 83.5009232,b 33.1966209,c 72.5719604,s 6,t 59,e1 0.0,e2 0.0,e3 0.0,e4 0.0,e5 0.0,e6 0.0}
DECL FDAT FP46={TOOL_NO 1,BASE_NO 0,IPO_FRAME #BASE}
DECL PDAT PPDAT46={VEL 100.0,ACC 100.0,APO_DIST 100.0}
DECL E6POS XP47={x 921.103577,y 127.618202,z 2039.95496,a -85.5017929,b 12.56493,c -33.684391,s 2,t 43,e1 0.0,e2 0.0,e3 0.0,e4 0.0,e5 0.0,e6 0.0}
DECL FDAT FP47={TOOL_NO 1,BASE_NO 0,IPO_FRAME #BASE}
DECL PDAT PPDAT47={VEL 100.0,ACC 100.0,APO_DIST 100.0}
DECL E6POS XP48={x 921.105713,y 346.04541,z 2035.99695,a -85.9543533,b -4.83763981,c -34.9262314,s 2,t 43,e1 0.0,e2 0.0,e3 0.0,e4 0.0,e5 0.0,e6 0.0}
DECL FDAT FP48={TOOL_NO 1,BASE_NO 0,IPO_FRAME #BASE}
DECL PDAT PPDAT48={VEL 100.0,ACC 100.0,APO_DIST 100.0}
DECL E6POS XP49={x 676.607727,y 443.065399,z 2411.16895,a -85.954689,b -4.83773804,c -34.9256897,s 2,t 43,e1 0.0,e2 0.0,e3 0.0,e4 0.0,e5 0.0,e6 0.0}
DECL FDAT FP49={TOOL_NO 1,BASE_NO 0,IPO_FRAME #BASE}
DECL PDAT PPDAT49={VEL 100.0,ACC 100.0,APO_DIST 100.0}
DECL E6POS XP50={x 676.614014,y 443.069397,z 2411.1731,a -77.9617386,b -35.9964294,c -138.580795,s 2,t 11,e1 0.0,e2 0.0,e3 0.0,e4 0.0,e5 0.0,e6 0.0}
DECL FDAT FP50={TOOL_NO 1,BASE_NO 0,IPO_FRAME #BASE}
DECL PDAT PPDAT50={VEL 100.0,ACC 100.0,APO_DIST 100.0}
DECL E6POS XP51={x 676.571411,y 442.991486,z 2411.2041,a -81.1397781,b 8.66814327,c -136.777298,s 2,t 11,e1 0.0,e2 0.0,e3 0.0,e4 0.0,e5 0.0,e6 0.0}
DECL FDAT FP51={TOOL_NO 1,BASE_NO 0,IPO_FRAME #BASE}
DECL PDAT PPDAT51={VEL 100.0,ACC 100.0,APO_DIST 100.0}
DECL E6POS XP52={x 422.825592,y 419.188599,z 2219.46899,a -81.1445618,b 8.66573238,c -136.781494,s 2,t 11,e1 0.0,e2 0.0,e3 0.0,e4 0.0,e5 0.0,e6 0.0}
DECL FDAT FP52={TOOL_NO 1,BASE_NO 0,IPO_FRAME #BASE}
DECL PDAT PPDAT52={VEL 100.0,ACC 100.0,APO_DIST 100.0}
DECL E6POS XP53={x 422.964386,y 419.113403,z 2219.50806,a -75.6708679,b 8.66452217,c -136.768799,s 2,t 11,e1 0.0,e2 0.0,e3 0.0,e4 0.0,e5 0.0,e6 0.0}
DECL FDAT FP53={TOOL_NO 1,BASE_NO 0,IPO_FRAME #BASE}
DECL PDAT PPDAT53={VEL 100.0,ACC 100.0,APO_DIST 100.0}
DECL E6POS XP54={x 597.503479,y 444.580414,z 2219.48999,a -75.6644897,b 8.66280556,c -136.776596,s 2,t 11,e1 0.0,e2 0.0,e3 0.0,e4 0.0,e5 0.0,e6 0.0}
DECL FDAT FP54={TOOL_NO 1,BASE_NO 0,IPO_FRAME #BASE}
DECL PDAT PPDAT54={VEL 100.0,ACC 100.0,APO_DIST 100.0}
DECL E6POS XP55={x 534.892273,y 417.391602,z 2290.5979,a -81.1428833,b 10.46803,c -137.775696,s 2,t 11,e1 0.0,e2 0.0,e3 0.0,e4 0.0,e5 0.0,e6 0.0}
DECL FDAT FP55={TOOL_NO 1,BASE_NO 0,IPO_FRAME #BASE}
DECL PDAT PPDAT55={VEL 100.0,ACC 100.0,APO_DIST 100.0}
DECL E6POS XP56={x -492.057098,y 376.424591,z 1439.44104,a 30.39114,b -23.5063496,c 172.467102,s 2,t 11,e1 0.0,e2 0.0,e3 0.0,e4 0.0,e5 0.0,e6 0.0}
DECL FDAT FP56={TOOL_NO 1,BASE_NO 0,IPO_FRAME #BASE}
DECL PDAT PPDAT56={VEL 100.0,ACC 100.0,APO_DIST 100.0}
DECL E6POS XP57={x -394.850006,y 526.049377,z 1686.42798,a 128.136703,b 79.5226974,c 88.2325134,s 6,t 27,e1 0.0,e2 0.0,e3 0.0,e4 0.0,e5 0.0,e6 0.0}
DECL FDAT FP57={TOOL_NO 1,BASE_NO 0,IPO_FRAME #BASE}
DECL PDAT PPDAT57={VEL 100.0,ACC 100.0,APO_DIST 100.0}
DECL E6POS XP58={x -394.840515,y 526.045227,z 2503.67896,a 128.140198,b 79.5215683,c 88.2362366,s 6,t 27,e1 0.0,e2 0.0,e3 0.0,e4 0.0,e5 0.0,e6 0.0}
DECL FDAT FP58={TOOL_NO 1,BASE_NO 0,IPO_FRAME #BASE}
DECL PDAT PPDAT58={VEL 100.0,ACC 100.0,APO_DIST 100.0}
DECL E6POS XP59={x 606.985718,y 526.04303,z 2503.68188,a 128.138504,b 79.5218735,c 88.2345123,s 6,t 27,e1 0.0,e2 0.0,e3 0.0,e4 0.0,e5 0.0,e6 0.0}
DECL FDAT FP59={TOOL_NO 1,BASE_NO 0,IPO_FRAME #BASE}
DECL PDAT PPDAT59={VEL 100.0,ACC 100.0,APO_DIST 100.0}
DECL E6POS XP60={x 606.984924,y -90.7351532,z 2503.68311,a 128.138794,b 79.5228424,c 88.2352371,s 6,t 26,e1 0.0,e2 0.0,e3 0.0,e4 0.0,e5 0.0,e6 0.0}
DECL FDAT FP60={TOOL_NO 1,BASE_NO 0,IPO_FRAME #BASE}
DECL PDAT PPDAT60={VEL 100.0,ACC 100.0,APO_DIST 100.0}
DECL E6POS XP61={x 606.976074,y -90.7321396,z 2424.72412,a 128.139603,b 79.523613,c 88.2362366,s 6,t 26,e1 0.0,e2 0.0,e3 0.0,e4 0.0,e5 0.0,e6 0.0}
DECL FDAT FP61={TOOL_NO 1,BASE_NO 0,IPO_FRAME #BASE}
DECL PDAT PPDAT61={VEL 100.0,ACC 100.0,APO_DIST 100.0}
DECL E6POS XP62={x 607.089478,y -90.8658066,z 2424.84106,a 118.763,b 79.5206985,c 88.090477,s 6,t 26,e1 0.0,e2 0.0,e3 0.0,e4 0.0,e5 0.0,e6 0.0}
DECL FDAT FP62={TOOL_NO 1,BASE_NO 0,IPO_FRAME #BASE}
DECL PDAT PPDAT62={VEL 100.0,ACC 100.0,APO_DIST 100.0}
DECL E6POS XP63={x 606.998596,y -90.7075119,z 2481.4209,a 100.4935,b 79.5218506,c 87.9541168,s 6,t 26,e1 0.0,e2 0.0,e3 0.0,e4 0.0,e5 0.0,e6 0.0}
DECL FDAT FP63={TOOL_NO 1,BASE_NO 0,IPO_FRAME #BASE}
DECL PDAT PPDAT63={VEL 100.0,ACC 100.0,APO_DIST 100.0}
DECL E6POS XP64={x 607.284912,y -91.0709534,z 2481.54492,a -129.107697,b 51.3308907,c -149.9953,s 6,t 26,e1 0.0,e2 0.0,e3 0.0,e4 0.0,e5 0.0,e6 0.0}
DECL FDAT FP64={TOOL_NO 1,BASE_NO 0,IPO_FRAME #BASE}
DECL PDAT PPDAT64={VEL 100.0,ACC 100.0,APO_DIST 100.0}
DECL E6POS XP65={x 607.261719,y 20.6743298,z 2306.62109,a -129.069107,b 51.3366013,c -149.983398,s 6,t 26,e1 0.0,e2 0.0,e3 0.0,e4 0.0,e5 0.0,e6 0.0}
DECL FDAT FP65={TOOL_NO 1,BASE_NO 0,IPO_FRAME #BASE}
DECL PDAT PPDAT65={VEL 100.0,ACC 100.0,APO_DIST 100.0}
DECL E6POS XP66={x 607.301086,y 325.022705,z 2227.7019,a -129.052994,b 51.3389702,c -149.972397,s 6,t 27,e1 0.0,e2 0.0,e3 0.0,e4 0.0,e5 0.0,e6 0.0}
DECL FDAT FP66={TOOL_NO 1,BASE_NO 0,IPO_FRAME #BASE}
DECL PDAT PPDAT66={VEL 100.0,ACC 100.0,APO_DIST 100.0}
DECL E6POS XP67={x 352.783813,y -270.055908,z 1490.54004,a 147.147705,b -38.4752083,c -172.865906,s 6,t 26,e1 0.0,e2 0.0,e3 0.0,e4 0.0,e5 0.0,e6 0.0}
DECL FDAT FP67={TOOL_NO 1,BASE_NO 0,IPO_FRAME #BASE}
DECL PDAT PPDAT67={VEL 100.0,ACC 100.0,APO_DIST 100.0}
DECL E6POS XP68={x 722.677795,y -474.232788,z 1611.09998,a 9.59308529,b -64.2729187,c 139.537506,s 2,t 10,e1 0.0,e2 0.0,e3 0.0,e4 0.0,e5 0.0,e6 0.0}
DECL FDAT FP68={TOOL_NO 1,BASE_NO 0,IPO_FRAME #BASE}
DECL PDAT PPDAT68={VEL 100.0,ACC 100.0,APO_DIST 100.0}
DECL E6POS XP69={x 514.347778,y -313.306793,z 1969.57202,a -34.9153404,b -1.72952497,c -3.7150991,s 2,t 10,e1 0.0,e2 0.0,e3 0.0,e4 0.0,e5 0.0,e6 0.0}
DECL FDAT FP69={TOOL_NO 1,BASE_NO 0,IPO_FRAME #BASE}
DECL PDAT PPDAT69={VEL 100.0,ACC 100.0,APO_DIST 100.0}
DECL E6POS XP70={x 519.878113,y -315.837494,z 2248.73511,a -36.0719795,b -3.73190999,c -3.76728797,s 2,t 10,e1 0.0,e2 0.0,e3 0.0,e4 0.0,e5 0.0,e6 0.0}
DECL FDAT FP70={TOOL_NO 1,BASE_NO 0,IPO_FRAME #BASE}
DECL PDAT PPDAT70={VEL 100.0,ACC 100.0,APO_DIST 100.0}
DECL E6POS XP71={x 519.881775,y -277.122589,z 2467.38696,a -36.0726013,b -3.73140192,c -3.76694489,s 2,t 10,e1 0.0,e2 0.0,e3 0.0,e4 0.0,e5 0.0,e6 0.0}
DECL FDAT FP71={TOOL_NO 1,BASE_NO 0,IPO_FRAME #BASE}
DECL PDAT PPDAT71={VEL 100.0,ACC 100.0,APO_DIST 100.0}
DECL E6POS XP72={x 519.562195,y -277.207214,z 2467.43896,a 26.0314808,b 26.1257706,c 139.365402,s 2,t 10,e1 0.0,e2 0.0,e3 0.0,e4 0.0,e5 0.0,e6 0.0}
DECL FDAT FP72={TOOL_NO 1,BASE_NO 0,IPO_FRAME #BASE}
DECL PDAT PPDAT72={VEL 100.0,ACC 100.0,APO_DIST 100.0}
DECL E6POS XP73={x 873.721375,y -87.1433411,z 1642.00903,a 83.546463,b -1.33227396,c 91.4121017,s 6,t 58,e1 0.0,e2 0.0,e3 0.0,e4 0.0,e5 0.0,e6 0.0}
DECL FDAT FP73={TOOL_NO 1,BASE_NO 0,IPO_FRAME #BASE}
DECL PDAT PPDAT73={VEL 100.0,ACC 100.0,APO_DIST 100.0}
DECL E6POS XP74={x 873.719727,y -87.1433868,z 1642.00195,a 86.3969269,b 63.3656311,c 93.1515427,s 6,t 26,e1 0.0,e2 0.0,e3 0.0,e4 0.0,e5 0.0,e6 0.0}
DECL FDAT FP74={TOOL_NO 1,BASE_NO 0,IPO_FRAME #BASE}
DECL PDAT PPDAT74={VEL 100.0,ACC 100.0,APO_DIST 100.0}
DECL E6POS XP75={x 873.718079,y -87.1432419,z 1641.995,a -98.2571564,b 52.4212799,c -92.3167267,s 6,t 58,e1 0.0,e2 0.0,e3 0.0,e4 0.0,e5 0.0,e6 0.0}
DECL FDAT FP75={TOOL_NO 1,BASE_NO 0,IPO_FRAME #BASE}
DECL PDAT PPDAT75={VEL 100.0,ACC 100.0,APO_DIST 100.0}
DECL E6POS XP76={x 873.486023,y -86.7437515,z 1634.81995,a -100.1511,b 52.3495598,c -94.8069382,s 6,t 58,e1 0.0,e2 0.0,e3 0.0,e4 0.0,e5 0.0,e6 0.0}
DECL FDAT FP76={TOOL_NO 1,BASE_NO 0,IPO_FRAME #BASE}
DECL PDAT PPDAT76={VEL 100.0,ACC 100.0,APO_DIST 100.0}
DECL E6POS XP77={x 896.842529,y -89.011467,z 1841.00806,a -102.858101,b 52.1103287,c -98.2126694,s 6,t 58,e1 0.0,e2 0.0,e3 0.0,e4 0.0,e5 0.0,e6 0.0}
DECL FDAT FP77={TOOL_NO 1,BASE_NO 0,IPO_FRAME #BASE}
DECL PDAT PPDAT77={VEL 100.0,ACC 100.0,APO_DIST 100.0}
DECL E6POS XP78={x 897.703918,y -83.4555435,z 1844.70105,a -91.8203964,b -38.1400604,c -95.4049377,s 6,t 58,e1 0.0,e2 0.0,e3 0.0,e4 0.0,e5 0.0,e6 0.0}
DECL FDAT FP78={TOOL_NO 1,BASE_NO 0,IPO_FRAME #BASE}
DECL PDAT PPDAT78={VEL 100.0,ACC 100.0,APO_DIST 100.0}
DECL E6POS XP79={x 529.078918,y -22.1784706,z 2112.57104,a 61.040451,b -3.74773407,c -23.0776691,s 2,t 42,e1 0.0,e2 0.0,e3 0.0,e4 0.0,e5 0.0,e6 0.0}
DECL FDAT FP79={TOOL_NO 1,BASE_NO 0,IPO_FRAME #BASE}
DECL PDAT PPDAT79={VEL 100.0,ACC 100.0,APO_DIST 100.0}
DECL E6POS XP80={x 527.087585,y 190.428406,z 1873.69897,a -152.824005,b -68.5615463,c 84.7780533,s 6,t 50,e1 0.0,e2 0.0,e3 0.0,e4 0.0,e5 0.0,e6 0.0}
DECL FDAT FP80={TOOL_NO 1,BASE_NO 0,IPO_FRAME #BASE}
DECL PDAT PPDAT80={VEL 100.0,ACC 100.0,APO_DIST 100.0}
DECL E6POS XP81={x 482.422791,y -285.181,z 1878.67798,a -28.0757408,b -59.2589493,c 84.1972885,s 2,t 34,e1 0.0,e2 0.0,e3 0.0,e4 0.0,e5 0.0,e6 0.0}
DECL FDAT FP81={TOOL_NO 1,BASE_NO 0,IPO_FRAME #BASE}
DECL PDAT PPDAT81={VEL 100.0,ACC 100.0,APO_DIST 100.0}
DECL E6POS XP82={x 521.025696,y -94.4028015,z 2109.44604,a -122.081596,b 19.6648693,c 15.7434902,s 6,t 50,e1 0.0,e2 0.0,e3 0.0,e4 0.0,e5 0.0,e6 0.0}
DECL FDAT FP82={TOOL_NO 1,BASE_NO 0,IPO_FRAME #BASE}
DECL PDAT PPDAT82={VEL 100.0,ACC 100.0,APO_DIST 100.0}
DECL E6POS XP83={x 899.490723,y -63.358799,z 1861.33105,a 91.2263107,b 71.0515976,c 92.2264328,s 2,t 34,e1 0.0,e2 0.0,e3 0.0,e4 0.0,e5 0.0,e6 0.0}
DECL FDAT FP83={TOOL_NO 1,BASE_NO 0,IPO_FRAME #BASE}
DECL PDAT PPDAT83={VEL 100.0,ACC 100.0,APO_DIST 100.0}
DECL E6POS XP84={x 406.722687,y -25.6750202,z 1427.052,a 84.8558502,b -3.53592896,c -131.892502,s 2,t 42,e1 0.0,e2 0.0,e3 0.0,e4 0.0,e5 0.0,e6 0.0}
DECL FDAT FP84={TOOL_NO 1,BASE_NO 0,IPO_FRAME #BASE}
DECL PDAT PPDAT84={VEL 100.0,ACC 100.0,APO_DIST 100.0}
DECL E6POS XP85={x -138.050995,y 6.55937576,z 3012.75098,a 85.7713623,b -1.02211297,c -17.0015106,s 7,t 58,e1 0.0,e2 0.0,e3 0.0,e4 0.0,e5 0.0,e6 0.0}
DECL FDAT FP85={TOOL_NO 1,BASE_NO 0,IPO_FRAME #BASE}
DECL PDAT PPDAT85={VEL 100.0,ACC 100.0,APO_DIST 100.0}
DECL E6POS XP86={x -99.3583603,y 7.66604519,z 2985.60693,a 83.9711227,b -1.02363098,c -17.0492096,s 7,t 58,e1 0.0,e2 0.0,e3 0.0,e4 0.0,e5 0.0,e6 0.0}
DECL FDAT FP86={TOOL_NO 1,BASE_NO 0,IPO_FRAME #BASE}
DECL PDAT PPDAT86={VEL 100.0,ACC 100.0,APO_DIST 100.0}
DECL E6POS XP87={x 752.619812,y -134.623703,z 2353.70093,a 81.146492,b -4.61759281,c 94.9607162,s 2,t 42,e1 0.0,e2 0.0,e3 0.0,e4 0.0,e5 0.0,e6 0.0}
DECL FDAT FP87={TOOL_NO 1,BASE_NO 0,IPO_FRAME #BASE}
DECL PDAT PPDAT87={VEL 100.0,ACC 100.0,APO_DIST 100.0}
DECL E6POS XP88={x 752.646973,y -134.378403,z 2464.69409,a 108.013603,b -4.68132019,c -17.5918808,s 2,t 34,e1 0.0,e2 0.0,e3 0.0,e4 0.0,e5 0.0,e6 0.0}
DECL FDAT FP88={TOOL_NO 1,BASE_NO 0,IPO_FRAME #BASE}
DECL PDAT PPDAT88={VEL 100.0,ACC 100.0,APO_DIST 100.0}
DECL E6POS XP89={x 752.455078,y -134.361206,z 2464.74512,a 120.274399,b 52.3513489,c 8.71092701,s 2,t 34,e1 0.0,e2 0.0,e3 0.0,e4 0.0,e5 0.0,e6 0.0}
DECL FDAT FP89={TOOL_NO 1,BASE_NO 0,IPO_FRAME #BASE}
DECL PDAT PPDAT89={VEL 100.0,ACC 100.0,APO_DIST 100.0}
DECL E6POS XP90={x 752.525513,y -134.267395,z 2464.6499,a 92.2309113,b -18.0458603,c 58.0951881,s 2,t 34,e1 0.0,e2 0.0,e3 0.0,e4 0.0,e5 0.0,e6 0.0}
DECL FDAT FP90={TOOL_NO 1,BASE_NO 0,IPO_FRAME #BASE}
DECL PDAT PPDAT90={VEL 100.0,ACC 100.0,APO_DIST 100.0}
DECL E6POS XP91={x 752.622803,y -114.498802,z 2414.7959,a 92.2273788,b -18.0442009,c 58.091629,s 2,t 34,e1 0.0,e2 0.0,e3 0.0,e4 0.0,e5 0.0,e6 0.0}
DECL FDAT FP91={TOOL_NO 1,BASE_NO 0,IPO_FRAME #BASE}
DECL PDAT PPDAT91={VEL 100.0,ACC 100.0,APO_DIST 100.0}
DECL E6POS XP92={x 815.588928,y -114.474602,z 2562.78296,a 95.1544418,b -17.5317097,c 50.5073814,s 2,t 34,e1 0.0,e2 0.0,e3 0.0,e4 0.0,e5 0.0,e6 0.0}
DECL FDAT FP92={TOOL_NO 1,BASE_NO 0,IPO_FRAME #BASE}
DECL PDAT PPDAT92={VEL 100.0,ACC 100.0,APO_DIST 100.0}
DECL E6POS XP93={x 13.2084198,y 9.55552483,z 3070.78711,a 161.808395,b -1.62972999,c 1.78704202,s 2,t 35,e1 0.0,e2 0.0,e3 0.0,e4 0.0,e5 0.0,e6 0.0}
DECL FDAT FP93={TOOL_NO 1,BASE_NO 0,IPO_FRAME #BASE}
DECL PDAT PPDAT93={VEL 100.0,ACC 100.0,APO_DIST 100.0}
DECL E6POS XP94={x -128.487305,y -220.863403,z 2730.3479,a -34.2470589,b -13.97542,c 105.6502,s 6,t 51,e1 0.0,e2 0.0,e3 0.0,e4 0.0,e5 0.0,e6 0.0}
DECL FDAT FP94={TOOL_NO 1,BASE_NO 0,IPO_FRAME #BASE}
DECL PDAT PPDAT94={VEL 100.0,ACC 100.0,APO_DIST 100.0}
DECL E6POS XP95={x 17.5380898,y 219.019196,z 2638.427,a 18.2083397,b -26.4088593,c -132.252701,s 2,t 43,e1 0.0,e2 0.0,e3 0.0,e4 0.0,e5 0.0,e6 0.0}
DECL FDAT FP95={TOOL_NO 1,BASE_NO 0,IPO_FRAME #BASE}
DECL PDAT PPDAT95={VEL 100.0,ACC 100.0,APO_DIST 100.0}
DECL E6POS XP96={x -196.500107,y -168.843002,z 2745.07202,a -39.3887596,b 38.6515999,c 105.390404,s 6,t 59,e1 0.0,e2 0.0,e3 0.0,e4 0.0,e5 0.0,e6 0.0}
DECL FDAT FP96={TOOL_NO 1,BASE_NO 0,IPO_FRAME #BASE}
DECL PDAT PPDAT96={VEL 100.0,ACC 100.0,APO_DIST 100.0}
DECL E6POS XP97={x -435.679108,y -456.34671,z 1616.25305,a -3.44279408,b -14.2607698,c -146.670807,s 5,t 63,e1 0.0,e2 0.0,e3 0.0,e4 0.0,e5 0.0,e6 0.0}
DECL FDAT FP97={TOOL_NO 1,BASE_NO 0,IPO_FRAME #BASE}
DECL PDAT PPDAT97={VEL 100.0,ACC 100.0,APO_DIST 100.0}
DECL E6POS XP98={x -349.021698,y -352.180695,z 1484.33704,a -6.94471502,b -21.6888599,c -135.380005,s 5,t 63,e1 0.0,e2 0.0,e3 0.0,e4 0.0,e5 0.0,e6 0.0}
DECL FDAT FP98={TOOL_NO 1,BASE_NO 0,IPO_FRAME #BASE}
DECL PDAT PPDAT98={VEL 100.0,ACC 100.0,APO_DIST 100.0}
DECL E6POS XP99={x -554.76709,y -356.133606,z 1834.40698,a -119.800003,b -29.4073009,c 43.1879501,s 1,t 47,e1 0.0,e2 0.0,e3 0.0,e4 0.0,e5 0.0,e6 0.0}
DECL FDAT FP99={TOOL_NO 1,BASE_NO 0,IPO_FRAME #BASE}
DECL PDAT PPDAT99={VEL 100.0,ACC 100.0,APO_DIST 100.0}
DECL E6POS XP100={x -437.045502,y -537.138184,z 1932.80396,a 99.1012268,b -1.29065895,c 0.955564678,s 5,t 55,e1 0.0,e2 0.0,e3 0.0,e4 0.0,e5 0.0,e6 0.0}
DECL FDAT FP100={TOOL_NO 1,BASE_NO 0,IPO_FRAME #BASE}
DECL PDAT PPDAT100={VEL 100.0,ACC 100.0,APO_DIST 100.0}
DECL E6POS XP101={x -443.991791,y -531.411499,z 1932.90906,a 98.2776108,b 0.137775198,c -0.310346812,s 5,t 55,e1 0.0,e2 0.0,e3 0.0,e4 0.0,e5 0.0,e6 0.0}
DECL FDAT FP101={TOOL_NO 1,BASE_NO 0,IPO_FRAME #BASE}
DECL PDAT PPDAT101={VEL 100.0,ACC 100.0,APO_DIST 100.0}
DECL E6POS XP102={x -443.959503,y -531.37262,z 1882.50696,a 98.2770233,b 0.144034505,c -0.302945703,s 5,t 55,e1 0.0,e2 0.0,e3 0.0,e4 0.0,e5 0.0,e6 0.0}
DECL FDAT FP102={TOOL_NO 1,BASE_NO 0,IPO_FRAME #BASE}
DECL PDAT PPDAT102={VEL 100.0,ACC 100.0,APO_DIST 100.0}
DECL E6POS XP103={x -443.95639,y -531.369629,z 2459.57397,a 98.2780304,b 0.144719005,c -0.301569909,s 5,t 55,e1 0.0,e2 0.0,e3 0.0,e4 0.0,e5 0.0,e6 0.0}
DECL FDAT FP103={TOOL_NO 1,BASE_NO 0,IPO_FRAME #BASE}
DECL PDAT PPDAT103={VEL 100.0,ACC 100.0,APO_DIST 100.0}
DECL E6POS XP104={x -205.858597,y -477.985504,z 2786.69312,a 105.819298,b 33.9970703,c 23.9303493,s 5,t 55,e1 0.0,e2 0.0,e3 0.0,e4 0.0,e5 0.0,e6 0.0}
DECL FDAT FP104={TOOL_NO 1,BASE_NO 0,IPO_FRAME #BASE}
DECL PDAT PPDAT104={VEL 100.0,ACC 100.0,APO_DIST 100.0}
DECL E6POS XP105={x 336.679413,y 53.0298309,z 2766.54199,a 109.7687,b 57.9234314,c 102.624901,s 6,t 51,e1 0.0,e2 0.0,e3 0.0,e4 0.0,e5 0.0,e6 0.0}
DECL FDAT FP105={TOOL_NO 1,BASE_NO 0,IPO_FRAME #BASE}
DECL PDAT PPDAT105={VEL 100.0,ACC 100.0,APO_DIST 100.0}
DECL E6POS XP106={x 661.836304,y -29.7462101,z 1598.55896,a 145.837296,b 2.915766,c 177.8293,s 6,t 50,e1 0.0,e2 0.0,e3 0.0,e4 0.0,e5 0.0,e6 0.0}
DECL FDAT FP106={TOOL_NO 1,BASE_NO 0,IPO_FRAME #BASE}
DECL PDAT PPDAT106={VEL 100.0,ACC 100.0,APO_DIST 100.0}
DECL E6POS XP107={x 991.485779,y -93.8970871,z 1923.90198,a 84.6064301,b 0.736399174,c 92.9489136,s 6,t 58,e1 0.0,e2 0.0,e3 0.0,e4 0.0,e5 0.0,e6 0.0}
DECL FDAT FP107={TOOL_NO 1,BASE_NO 0,IPO_FRAME #BASE}
DECL PDAT PPDAT107={VEL 100.0,ACC 100.0,APO_DIST 100.0}
DECL E6POS XP108={x 727.591125,y -76.0883713,z 3015.31104,a 40.80616,b -1.36277902,c 2.90668607,s 6,t 58,e1 0.0,e2 0.0,e3 0.0,e4 0.0,e5 0.0,e6 0.0}
DECL FDAT FP108={TOOL_NO 1,BASE_NO 0,IPO_FRAME #BASE}
DECL PDAT PPDAT108={VEL 100.0,ACC 100.0,APO_DIST 100.0}
DECL E6POS XP109={x 52.6107483,y -76.3511887,z 3158.91992,a 40.7964516,b -1.36811101,c 2.90851212,s 6,t 58,e1 0.0,e2 0.0,e3 0.0,e4 0.0,e5 0.0,e6 0.0}
DECL FDAT FP109={TOOL_NO 1,BASE_NO 0,IPO_FRAME #BASE}
DECL PDAT PPDAT109={VEL 100.0,ACC 100.0,APO_DIST 100.0}
DECL E6POS XP110={x 52.6367798,y -653.577881,z 3010.34595,a 40.7968407,b -1.37141001,c 2.9194119,s 6,t 50,e1 0.0,e2 0.0,e3 0.0,e4 0.0,e5 0.0,e6 0.0}
DECL FDAT FP110={TOOL_NO 1,BASE_NO 0,IPO_FRAME #BASE}
DECL PDAT PPDAT110={VEL 100.0,ACC 100.0,APO_DIST 100.0}
DECL E6POS XP111={x 52.6099091,y -653.457703,z 2670.83008,a 40.7954292,b -1.36951196,c 2.91018009,s 6,t 50,e1 0.0,e2 0.0,e3 0.0,e4 0.0,e5 0.0,e6 0.0}
DECL FDAT FP111={TOOL_NO 1,BASE_NO 0,IPO_FRAME #BASE}
DECL PDAT PPDAT111={VEL 100.0,ACC 100.0,APO_DIST 100.0}
DECL INT LAST_XP_POINT=579
DECL E6POS XP112={x 52.5952415,y -876.464417,z 1992.52905,a 58.9748688,b -1.362378,c 2.90494704,s 6,t 50,e1 0.0,e2 0.0,e3 0.0,e4 0.0,e5 0.0,e6 0.0}
DECL FDAT FP112={TOOL_NO 1,BASE_NO 0,IPO_FRAME #BASE}
DECL PDAT PPDAT112={VEL 100.0,ACC 100.0,APO_DIST 100.0}
DECL E6POS XP113={x -76.5833435,y 363.044006,z 3240.97705,a 59.0353813,b -1.41373599,c 2.88797498,s 6,t 27,e1 0.0,e2 0.0,e3 0.0,e4 0.0,e5 0.0,e6 0.0}
DECL FDAT FP113={TOOL_NO 1,BASE_NO 0,IPO_FRAME #BASE}
DECL PDAT PPDAT113={VEL 100.0,ACC 100.0,APO_DIST 100.0}
DECL E6POS XP114={x -1339.04297,y -48.73592,z 2099.98901,a -87.8156891,b 6.90914679,c 88.0969086,s 6,t 50,e1 0.0,e2 0.0,e3 0.0,e4 0.0,e5 0.0,e6 0.0}
DECL FDAT FP114={TOOL_NO 1,BASE_NO 0,IPO_FRAME #BASE}
DECL PDAT PPDAT114={VEL 100.0,ACC 100.0,APO_DIST 100.0}
DECL E6POS XP115={x 445.791992,y 13.6370401,z 3047.40894,a -94.1068802,b -3.23984408,c -31.2618408,s 5,t 54,e1 0.0,e2 0.0,e3 0.0,e4 0.0,e5 0.0,e6 0.0}
DECL FDAT FP115={TOOL_NO 1,BASE_NO 0,IPO_FRAME #BASE}
DECL PDAT PPDAT115={VEL 100.0,ACC 100.0,APO_DIST 100.0}
DECL E6POS XP116={x 622.982971,y 34.6125603,z 2762.38501,a -93.0572968,b -2.47985101,c 2.92759395,s 1,t 38,e1 0.0,e2 0.0,e3 0.0,e4 0.0,e5 0.0,e6 0.0}
DECL FDAT FP116={TOOL_NO 1,BASE_NO 0,IPO_FRAME #BASE}
DECL PDAT PPDAT116={VEL 100.0,ACC 100.0,APO_DIST 100.0}
DECL E6POS XP117={x 710.174622,y -63.8623505,z 1482.26001,a 85.9968796,b -0.728000879,c -178.896103,s 2,t 42,e1 0.0,e2 0.0,e3 0.0,e4 0.0,e5 0.0,e6 0.0}
DECL FDAT FP117={TOOL_NO 1,BASE_NO 0,IPO_FRAME #BASE}
DECL PDAT PPDAT117={VEL 100.0,ACC 100.0,APO_DIST 100.0}
DECL E6POS XP118={x 710.174622,y -63.8623505,z 1482.26001,a 85.9968796,b -0.728000879,c -178.896103,s 2,t 42,e1 0.0,e2 0.0,e3 0.0,e4 0.0,e5 0.0,e6 0.0}
DECL FDAT FP118={TOOL_NO 1,BASE_NO 0,IPO_FRAME #BASE}
DECL LDAT LCPDAT1={VEL 2.0,ACC 100.0,APO_DIST 100.0,APO_FAC 50.0}
DECL E6POS XP119={x 710.175476,y -1014.49103,z 1483.27502,a 85.9965591,b -0.727580488,c -178.896301,s 2,t 34,e1 0.0,e2 0.0,e3 0.0,e4 0.0,e5 0.0,e6 0.0}
DECL FDAT FP119={TOOL_NO 1,BASE_NO 0,IPO_FRAME #BASE}
DECL LDAT LCPDAT2={VEL 2.0,ACC 100.0,APO_DIST 100.0,APO_FAC 50.0}
DECL E6POS XP120={x 710.172485,y 1084.77295,z 1483.26794,a 85.9965363,b -0.727106512,c -178.895996,s 2,t 43,e1 0.0,e2 0.0,e3 0.0,e4 0.0,e5 0.0,e6 0.0}
DECL FDAT FP120={TOOL_NO 1,BASE_NO 0,IPO_FRAME #BASE}
DECL PDAT PPDAT118={VEL 100.0,ACC 100.0,APO_DIST 100.0}
DECL E6POS XP121={x -688.051819,y 1088.13,z 1483.276,a 85.9968033,b -0.727819622,c -178.895493,s 2,t 43,e1 0.0,e2 0.0,e3 0.0,e4 0.0,e5 0.0,e6 0.0}
DECL FDAT FP121={TOOL_NO 1,BASE_NO 0,IPO_FRAME #BASE}
DECL PDAT PPDAT119={VEL 100.0,ACC 100.0,APO_DIST 100.0}
DECL E6POS XP122={x -688.050903,y 1088.13196,z 2238.00488,a 85.9966965,b -0.727052629,c -178.895905,s 2,t 43,e1 0.0,e2 0.0,e3 0.0,e4 0.0,e5 0.0,e6 0.0}
DECL FDAT FP122={TOOL_NO 1,BASE_NO 0,IPO_FRAME #BASE}
DECL PDAT PPDAT120={VEL 100.0,ACC 100.0,APO_DIST 100.0}
DECL E6POS XP123={x -78.7586136,y 830.951782,z 2238.00806,a 85.997139,b -0.727514982,c -178.895493,s 2,t 43,e1 0.0,e2 0.0,e3 0.0,e4 0.0,e5 0.0,e6 0.0}
DECL FDAT FP123={TOOL_NO 1,BASE_NO 0,IPO_FRAME #BASE}
DECL PDAT PPDAT121={VEL 100.0,ACC 100.0,APO_DIST 100.0}
DECL E6POS XP124={x 696.539978,y 826.553284,z 2238.01001,a 85.9973831,b -0.727540374,c -178.896103,s 2,t 43,e1 0.0,e2 0.0,e3 0.0,e4 0.0,e5 0.0,e6 0.0}
DECL FDAT FP124={TOOL_NO 1,BASE_NO 0,IPO_FRAME #BASE}
DECL PDAT PPDAT122={VEL 100.0,ACC 100.0,APO_DIST 100.0}
DECL E6POS XP125={x 696.540222,y 826.55072,z 2238.01001,a 98.3100128,b 0.693525612,c 1.33698404,s 2,t 35,e1 0.0,e2 0.0,e3 0.0,e4 0.0,e5 0.0,e6 0.0}
DECL FDAT FP125={TOOL_NO 1,BASE_NO 0,IPO_FRAME #BASE}
DECL PDAT PPDAT123={VEL 100.0,ACC 100.0,APO_DIST 100.0}
DECL E6POS XP126={x 696.482422,y 826.485229,z 3002.65796,a 98.3093185,b 0.684386611,c 1.326756,s 2,t 35,e1 0.0,e2 0.0,e3 0.0,e4 0.0,e5 0.0,e6 0.0}
DECL FDAT FP126={TOOL_NO 1,BASE_NO 0,IPO_FRAME #BASE}
DECL PDAT PPDAT124={VEL 100.0,ACC 100.0,APO_DIST 100.0}
DECL E6POS XP127={x 199.969894,y -429.384308,z 3002.65503,a 98.3047791,b 0.688694775,c 1.32615101,s 2,t 34,e1 0.0,e2 0.0,e3 0.0,e4 0.0,e5 0.0,e6 0.0}
DECL FDAT FP127={TOOL_NO 1,BASE_NO 0,IPO_FRAME #BASE}
DECL PDAT PPDAT125={VEL 100.0,ACC 100.0,APO_DIST 100.0}
DECL E6POS XP128={x -918.844482,y -5.84095478,z 1909.37598,a 89.5914078,b 15.3547802,c -92.9045868,s 2,t 35,e1 0.0,e2 0.0,e3 0.0,e4 0.0,e5 0.0,e6 0.0}
DECL FDAT FP128={TOOL_NO 1,BASE_NO 0,IPO_FRAME #BASE}
DECL PDAT PPDAT126={VEL 100.0,ACC 100.0,APO_DIST 100.0}
DECL E6POS XP129={x 830.454102,y 5.31626797,z 2066.03394,a 90.4962769,b -15.37327,c 89.522583,s 1,t 39,e1 0.0,e2 0.0,e3 0.0,e4 0.0,e5 0.0,e6 0.0}
DECL FDAT FP129={TOOL_NO 1,BASE_NO 0,IPO_FRAME #BASE}
DECL PDAT PPDAT127={VEL 100.0,ACC 100.0,APO_DIST 100.0}
DECL E6POS XP130={x 1619.98499,y -0.161705703,z 2194.88892,a -140.350998,b 89.9749222,c -140.345306,s 2,t 2,e1 0.0,e2 0.0,e3 0.0,e4 0.0,e5 0.0,e6 0.0}
DECL FDAT FP130={TOOL_NO 1,BASE_NO 0,IPO_FRAME #BASE}
DECL PDAT PPDAT128={VEL 100.0,ACC 100.0,APO_DIST 100.0}
DECL E6POS XP131={x 1619.98499,y -0.161701694,z 2194.88892,a -140.269897,b 89.9749069,c -140.264206,s 2,t 2,e1 0.0,e2 0.0,e3 0.0,e4 0.0,e5 0.0,e6 0.0}
DECL FDAT FP131={TOOL_NO 1,BASE_NO 0,IPO_FRAME #BASE}
DECL PDAT PPDAT129={VEL 100.0,ACC 100.0,APO_DIST 100.0}
DECL E6POS XP132={x 1436.95398,y -1190.03296,z 1852.45105,a 122.7612,b 82.1193085,c 123.386497,s 2,t 10,e1 0.0,e2 0.0,e3 0.0,e4 0.0,e5 0.0,e6 0.0}
DECL E6POS XP133={x 1436.953,y 1035.35803,z 1852.43994,a 122.7658,b 82.1197281,c 123.391403,s 2,t 11,e1 0.0,e2 0.0,e3 0.0,e4 0.0,e5 0.0,e6 0.0}
DECL FDAT FP133={TOOL_NO 1,BASE_NO 0,IPO_FRAME #BASE}
DECL LDAT LCPDAT3={VEL 2.0,ACC 100.0,APO_DIST 100.0,APO_FAC 50.0}
DECL E6POS XP134={x 1619.98901,y -0.174462497,z 2194.78711,a -154.099106,b 89.9706116,c -154.093094,s 2,t 10,e1 0.0,e2 0.0,e3 0.0,e4 0.0,e5 0.0,e6 0.0}
DECL FDAT FP134={TOOL_NO 1,BASE_NO 0,IPO_FRAME #BASE}
DECL PDAT PPDAT130={VEL 100.0,ACC 100.0,APO_DIST 100.0}
DECL E6POS XP135={x 1208.875,y -812.839905,z 1585.56995,a -172.129807,b 89.9697189,c -172.127197,s 2,t 10,e1 0.0,e2 0.0,e3 0.0,e4 0.0,e5 0.0,e6 0.0}
DECL E6POS XP136={x 1208.86902,y 7.70442915,z 1585.56299,a -171.229004,b 89.9693985,c -171.226395,s 2,t 11,e1 0.0,e2 0.0,e3 0.0,e4 0.0,e5 0.0,e6 0.0}
DECL FDAT FP136={TOOL_NO 1,BASE_NO 0,IPO_FRAME #BASE}
DECL LDAT LCPDAT4={VEL 2.0,ACC 100.0,APO_DIST 100.0,APO_FAC 50.0}
DECL E6POS XP137={x 1101.78101,y 308.098694,z 1343.38,a 85.9301071,b -0.842971802,c -174.109695,s 2,t 43,e1 0.0,e2 0.0,e3 0.0,e4 0.0,e5 0.0,e6 0.0}
DECL E6POS XP138={x 1101.78796,y -300.667908,z 1343.38599,a 85.9297333,b -0.842814922,c -174.110397,s 2,t 34,e1 0.0,e2 0.0,e3 0.0,e4 0.0,e5 0.0,e6 0.0}
DECL FDAT FP138={TOOL_NO 1,BASE_NO 0,IPO_FRAME #BASE}
DECL LDAT LCPDAT5={VEL 2.0,ACC 100.0,APO_DIST 100.0,APO_FAC 50.0}
DECL E6POS XP139={x 676.888428,y -87.4530716,z 1379.58301,a 85.8759995,b -0.811197221,c -174.122192,s 2,t 42,e1 0.0,e2 0.0,e3 0.0,e4 0.0,e5 0.0,e6 0.0}
DECL FDAT FP139={TOOL_NO 1,BASE_NO 0,IPO_FRAME #BASE}
DECL PDAT PPDAT131={VEL 100.0,ACC 100.0,APO_DIST 100.0}
DECL E6POS XP140={x 718.616272,y -50.0314903,z 1789.96399,a 85.9308395,b -0.843019187,c -174.100204,s 2,t 42,e1 0.0,e2 0.0,e3 0.0,e4 0.0,e5 0.0,e6 0.0}
DECL FDAT FP140={TOOL_NO 1,BASE_NO 0,IPO_FRAME #BASE}
DECL PDAT PPDAT132={VEL 100.0,ACC 100.0,APO_DIST 100.0}
DECL E6POS XP141={x 718.616089,y 1273.56104,z 1789.96399,a 85.9307404,b -0.843725026,c -174.100006,s 2,t 43,e1 0.0,e2 0.0,e3 0.0,e4 0.0,e5 0.0,e6 0.0}
DECL FDAT FP141={TOOL_NO 1,BASE_NO 0,IPO_FRAME #BASE}
DECL LDAT LCPDAT6={VEL 2.0,ACC 100.0,APO_DIST 100.0,APO_FAC 50.0}
DECL E6POS XP142={x 718.619385,y -1284.73901,z 1789.974,a 85.9307709,b -0.843700707,c -174.100204,s 2,t 34,e1 0.0,e2 0.0,e3 0.0,e4 0.0,e5 0.0,e6 0.0}
DECL FDAT FP142={TOOL_NO 1,BASE_NO 0,IPO_FRAME #BASE}
DECL LDAT LCPDAT7={VEL 2.0,ACC 100.0,APO_DIST 100.0,APO_FAC 50.0}
DECL E6POS XP143={x -766.560913,y -1284.75403,z 1789.98303,a 85.9355927,b -0.84204942,c -174.101593,s 2,t 2,e1 0.0,e2 0.0,e3 0.0,e4 0.0,e5 0.0,e6 0.0}
DECL FDAT FP143={TOOL_NO 1,BASE_NO 0,IPO_FRAME #BASE}
DECL LDAT LCPDAT8={VEL 2.0,ACC 100.0,APO_DIST 100.0,APO_FAC 50.0}
DECL E6POS XP144={x -766.522583,y -36.58992,z 1789.995,a 85.937027,b -0.841355979,c -174.096405,s 2,t 2,e1 0.0,e2 0.0,e3 0.0,e4 0.0,e5 0.0,e6 0.0}
DECL FDAT FP144={TOOL_NO 1,BASE_NO 0,IPO_FRAME #BASE}
DECL LDAT LCPDAT9={VEL 2.0,ACC 100.0,APO_DIST 100.0,APO_FAC 50.0}
DECL E6POS XP145={x 384.592499,y -1408.48303,z 1790.00403,a 85.9372025,b -0.840705216,c -174.096603,s 2,t 34,e1 0.0,e2 0.0,e3 0.0,e4 0.0,e5 0.0,e6 0.0}
DECL FDAT FP145={TOOL_NO 1,BASE_NO 0,IPO_FRAME #BASE}
DECL LDAT LCPDAT10={VEL 2.0,ACC 100.0,APO_DIST 100.0,APO_FAC 50.0}
DECL E6POS XP146={x 598.668518,y 1375.28406,z 1790.04602,a 85.9391632,b -0.842212677,c -174.093002,s 2,t 43,e1 0.0,e2 0.0,e3 0.0,e4 0.0,e5 0.0,e6 0.0}
DECL FDAT FP146={TOOL_NO 1,BASE_NO 0,IPO_FRAME #BASE}
DECL LDAT LCPDAT11={VEL 2.0,ACC 100.0,APO_DIST 100.0,APO_FAC 50.0}
DECL E6POS XP147={x -1789.06396,y 363.775085,z 1790.047,a 85.9391632,b -0.842145383,c -174.092804,s 2,t 35,e1 0.0,e2 0.0,e3 0.0,e4 0.0,e5 0.0,e6 0.0}
DECL FDAT FP147={TOOL_NO 1,BASE_NO 0,IPO_FRAME #BASE}
DECL LDAT LCPDAT12={VEL 2.0,ACC 100.0,APO_DIST 100.0,APO_FAC 50.0}
DECL E6POS XP148={x 1619.99097,y -0.0378511809,z 2194.95508,a -122.182701,b 89.9861832,c -122.181396,s 2,t 2,e1 0.0,e2 0.0,e3 0.0,e4 0.0,e5 0.0,e6 0.0}
DECL FDAT FP148={TOOL_NO 1,BASE_NO 0,IPO_FRAME #BASE}
DECL PDAT PPDAT133={VEL 100.0,ACC 100.0,APO_DIST 100.0}
DECL E6POS XP149={x 99.0811005,y -0.00253095501,z 3198.14404,a -0.0130024599,b 1.49921203,c -0.000300739193,s 2,t 2,e1 0.0,e2 0.0,e3 0.0,e4 0.0,e5 0.0,e6 0.0}
DECL FDAT FP149={TOOL_NO 1,BASE_NO 0,IPO_FRAME #BASE}
DECL PDAT PPDAT134={VEL 100.0,ACC 100.0,APO_DIST 100.0}
DECL E6POS XP150={x -620.150574,y 0.0157987699,z 2086.74194,a -6.98730898,b -89.9051285,c 6.98583984,s 1,t 6,e1 0.0,e2 0.0,e3 0.0,e4 0.0,e5 0.0,e6 0.0}
DECL FDAT FP150={TOOL_NO 1,BASE_NO 0,IPO_FRAME #BASE}
DECL PDAT PPDAT135={VEL 100.0,ACC 100.0,APO_DIST 100.0}
DECL E6POS XP151={x -350.350586,y 0.0595526993,z 1816.29199,a -180.0,b -0.0424678102,c 179.989304,s 5,t 22,e1 0.0,e2 0.0,e3 0.0,e4 0.0,e5 0.0,e6 0.0}
DECL FDAT FP151={TOOL_NO 1,BASE_NO 0,IPO_FRAME #BASE}
DECL PDAT PPDAT136={VEL 100.0,ACC 100.0,APO_DIST 100.0}
DECL E6POS XP152={x -350.420593,y 0.0580656081,z 1812.22498,a 179.998306,b -0.0610494502,c 179.989304,s 5,t 54,e1 0.0,e2 0.0,e3 0.0,e4 0.0,e5 0.0,e6 0.0}
DECL FDAT FP152={TOOL_NO 1,BASE_NO 0,IPO_FRAME #BASE}
DECL PDAT PPDAT137={VEL 100.0,ACC 100.0,APO_DIST 100.0}
DECL E6POS XP153={x -1028.41394,y 0.0640567467,z 1812.10706,a 179.998398,b -0.0444437191,c 179.989197,s 5,t 22,e1 0.0,e2 0.0,e3 0.0,e4 0.0,e5 0.0,e6 0.0}
DECL FDAT FP153={TOOL_NO 1,BASE_NO 0,IPO_FRAME #BASE}
DECL PDAT PPDAT138={VEL 100.0,ACC 100.0,APO_DIST 100.0}
DECL E6POS XP154={x -840.15332,y 0.0595172495,z 1030.40002,a 179.997406,b -0.0750442892,c 179.990005,s 5,t 54,e1 0.0,e2 0.0,e3 0.0,e4 0.0,e5 0.0,e6 0.0}
DECL FDAT FP154={TOOL_NO 1,BASE_NO 0,IPO_FRAME #BASE}
DECL PDAT PPDAT139={VEL 100.0,ACC 100.0,APO_DIST 100.0}
DECL E6POS XP155={x -598.344299,y 0.0649362728,z 1179.56104,a 179.965103,b 63.4142113,c 179.957596,s 5,t 54,e1 0.0,e2 0.0,e3 0.0,e4 0.0,e5 0.0,e6 0.0}
DECL FDAT FP155={TOOL_NO 1,BASE_NO 0,IPO_FRAME #BASE}
DECL PDAT PPDAT140={VEL 100.0,ACC 100.0,APO_DIST 100.0}
DECL E6POS XP156={x 700.694885,y -0.0667810887,z 1384.79004,a 179.721298,b -86.9002838,c -179.710602,s 2,t 34,e1 0.0,e2 0.0,e3 0.0,e4 0.0,e5 0.0,e6 0.0}
DECL FDAT FP156={TOOL_NO 1,BASE_NO 0,IPO_FRAME #BASE}
DECL PDAT PPDAT141={VEL 100.0,ACC 100.0,APO_DIST 100.0}
DECL E6POS XP157={x 105.960403,y 0.0282347109,z 3056.28491,a -91.6419678,b 0.161802694,c 5.66286898,s 1,t 39,e1 0.0,e2 0.0,e3 0.0,e4 0.0,e5 0.0,e6 0.0}
DECL FDAT FP157={TOOL_NO 1,BASE_NO 0,IPO_FRAME #BASE}
DECL PDAT PPDAT142={VEL 100.0,ACC 100.0,APO_DIST 100.0}
DECL E6POS XP158={x 909.859009,y 0.171782106,z 1801.67004,a -91.6433334,b 0.102886103,c 3.6484921,s 1,t 39,e1 0.0,e2 0.0,e3 0.0,e4 0.0,e5 0.0,e6 0.0}
DECL FDAT FP158={TOOL_NO 1,BASE_NO 0,IPO_FRAME #BASE}
DECL PDAT PPDAT143={VEL 100.0,ACC 100.0,APO_DIST 100.0}
DECL E6POS XP159={x 909.784485,y -313.817505,z 2461.67212,a -91.6422424,b 0.102985598,c 3.65116501,s 1,t 47,e1 0.0,e2 0.0,e3 0.0,e4 0.0,e5 0.0,e6 0.0}
DECL FDAT FP159={TOOL_NO 1,BASE_NO 0,IPO_FRAME #BASE}
DECL PDAT PPDAT144={VEL 100.0,ACC 100.0,APO_DIST 100.0}
DECL E6POS XP160={x 193.210007,y 402.010315,z 3260.04297,a 172.193802,b -0.0234979093,c 0.075235717,s 0,t 43,e1 0.0,e2 0.0,e3 0.0,e4 0.0,e5 0.0,e6 0.0}
DECL FDAT FP160={TOOL_NO 1,BASE_NO 0,IPO_FRAME #BASE}
DECL PDAT PPDAT145={VEL 100.0,ACC 100.0,APO_DIST 100.0}
DECL E6POS XP161={x 880.489319,y 933.132324,z 3121.42603,a 153.342804,b -6.48646116,c 20.6594791,s 0,t 43,e1 0.0,e2 0.0,e3 0.0,e4 0.0,e5 0.0,e6 0.0}
DECL FDAT FP161={TOOL_NO 1,BASE_NO 0,IPO_FRAME #BASE}
DECL PDAT PPDAT146={VEL 100.0,ACC 100.0,APO_DIST 100.0}
DECL E6POS XP162={x -686.627808,y -727.668396,z 2694.28003,a 150.545807,b 11.3533497,c -38.5334396,s 1,t 43,e1 0.0,e2 0.0,e3 0.0,e4 0.0,e5 0.0,e6 0.0}
DECL FDAT FP162={TOOL_NO 1,BASE_NO 0,IPO_FRAME #BASE}
DECL PDAT PPDAT147={VEL 100.0,ACC 100.0,APO_DIST 100.0}
DECL E6POS XP163={x -992.755188,y 124.052597,z 2694.28394,a 96.7610779,b 11.3532896,c -38.5331993,s 1,t 42,e1 0.0,e2 0.0,e3 0.0,e4 0.0,e5 0.0,e6 0.0}
DECL FDAT FP163={TOOL_NO 1,BASE_NO 0,IPO_FRAME #BASE}
DECL PDAT PPDAT148={VEL 100.0,ACC 100.0,APO_DIST 100.0}
DECL E6POS XP164={x 409.92569,y 912.637512,z 2694.28589,a -10.30406,b 11.3534203,c -38.5330811,s 1,t 42,e1 0.0,e2 0.0,e3 0.0,e4 0.0,e5 0.0,e6 0.0}
DECL FDAT FP164={TOOL_NO 1,BASE_NO 0,IPO_FRAME #BASE}
DECL PDAT PPDAT149={VEL 100.0,ACC 100.0,APO_DIST 100.0}
DECL E6POS XP165={x 1000.46301,y -0.678283393,z 2694.29492,a -76.1545334,b 11.3534698,c -38.5323906,s 1,t 42,e1 0.0,e2 0.0,e3 0.0,e4 0.0,e5 0.0,e6 0.0}
DECL FDAT FP165={TOOL_NO 1,BASE_NO 0,IPO_FRAME #BASE}
DECL PDAT PPDAT150={VEL 100.0,ACC 100.0,APO_DIST 100.0}
DECL E6POS XP166={x 927.409912,y -0.628985107,z 2755.93091,a -75.6971207,b 10.7653704,c -36.1489487,s 1,t 42,e1 0.0,e2 0.0,e3 0.0,e4 0.0,e5 0.0,e6 0.0}
DECL FDAT FP166={TOOL_NO 1,BASE_NO 0,IPO_FRAME #BASE}
DECL PDAT PPDAT151={VEL 100.0,ACC 100.0,APO_DIST 100.0}
DECL E6POS XP167={x 1594.672,y -147.282806,z 1830.703,a 84.8937683,b 26.0698605,c 90.9309464,s 6,t 58,e1 0.0,e2 0.0,e3 0.0,e4 0.0,e5 0.0,e6 0.0}
DECL FDAT FP167={TOOL_NO 1,BASE_NO 0,IPO_FRAME #BASE}
DECL PDAT PPDAT152={VEL 100.0,ACC 100.0,APO_DIST 100.0}
DECL E6POS XP168={x 1849.31995,y -147.290207,z 1830.69202,a 84.8936462,b 26.0701199,c 90.931221,s 6,t 58,e1 0.0,e2 0.0,e3 0.0,e4 0.0,e5 0.0,e6 0.0}
DECL FDAT FP168={TOOL_NO 1,BASE_NO 0,IPO_FRAME #BASE}
DECL PDAT PPDAT153={VEL 100.0,ACC 100.0,APO_DIST 100.0}
DECL E6POS XP169={x 909.749023,y -147.290894,z 1830.91003,a 84.8774033,b 26.0414391,c 90.9037704,s 6,t 50,e1 0.0,e2 0.0,e3 0.0,e4 0.0,e5 0.0,e6 0.0}
DECL FDAT FP169={TOOL_NO 1,BASE_NO 0,IPO_FRAME #BASE}
DECL PDAT PPDAT154={VEL 100.0,ACC 100.0,APO_DIST 100.0}
DECL E6POS XP170={x 1754.26697,y -147.109497,z 1831.02698,a 84.8834,b 26.0403004,c 90.8913879,s 6,t 58,e1 0.0,e2 0.0,e3 0.0,e4 0.0,e5 0.0,e6 0.0}
DECL FDAT FP170={TOOL_NO 1,BASE_NO 0,IPO_FRAME #BASE}
DECL PDAT PPDAT155={VEL 100.0,ACC 100.0,APO_DIST 100.0}
DECL E6POS XP171={x 900.760071,y -147.053497,z 1831.17297,a 84.8804092,b 26.0369606,c 90.8772964,s 6,t 50,e1 0.0,e2 0.0,e3 0.0,e4 0.0,e5 0.0,e6 0.0}
DECL FDAT FP171={TOOL_NO 1,BASE_NO 0,IPO_FRAME #BASE}
DECL PDAT PPDAT156={VEL 100.0,ACC 100.0,APO_DIST 100.0}
DECL E6POS XP172={x 1831.729,y -147.057007,z 1831.17102,a 84.8804398,b 26.0372906,c 90.8773727,s 6,t 58,e1 0.0,e2 0.0,e3 0.0,e4 0.0,e5 0.0,e6 0.0}
DECL FDAT FP172={TOOL_NO 1,BASE_NO 0,IPO_FRAME #BASE}
DECL PDAT PPDAT157={VEL 100.0,ACC 100.0,APO_DIST 100.0}
DECL E6POS XP173={x 22.1363697,y 1947.67603,z 1801.41602,a -73.0717468,b 89.9894638,c -162.288895,s 6,t 27,e1 0.0,e2 0.0,e3 0.0,e4 0.0,e5 0.0,e6 0.0}
DECL FDAT FP173={TOOL_NO 1,BASE_NO 0,IPO_FRAME #BASE}
DECL PDAT PPDAT158={VEL 100.0,ACC 100.0,APO_DIST 100.0}
DECL E6POS XP174={x 22.1354904,y 1947.66602,z 543.987122,a -72.872467,b 89.9886703,c -162.089706,s 6,t 27,e1 0.0,e2 0.0,e3 0.0,e4 0.0,e5 0.0,e6 0.0}
DECL FDAT FP174={TOOL_NO 1,BASE_NO 0,IPO_FRAME #BASE}
DECL PDAT PPDAT159={VEL 100.0,ACC 100.0,APO_DIST 100.0}
DECL E6POS XP175={x 63.0649109,y 1808.63501,z 103.495499,a -92.3154831,b -2.39625597,c 179.993301,s 2,t 43,e1 0.0,e2 0.0,e3 0.0,e4 0.0,e5 0.0,e6 0.0}
DECL FDAT FP175={TOOL_NO 1,BASE_NO 0,IPO_FRAME #BASE}
DECL PDAT PPDAT160={VEL 100.0,ACC 100.0,APO_DIST 100.0}
DECL E6POS XP176={x 63.0495415,y 1808.48901,z 2110.69189,a -92.3198624,b -2.36630106,c 179.993607,s 2,t 43,e1 0.0,e2 0.0,e3 0.0,e4 0.0,e5 0.0,e6 0.0}
DECL FDAT FP176={TOOL_NO 1,BASE_NO 0,IPO_FRAME #BASE}
DECL PDAT PPDAT161={VEL 100.0,ACC 100.0,APO_DIST 100.0}
DECL E6POS XP177={x 63.0451508,y 1808.46997,z -0.613860071,a -92.3198318,b -2.36753607,c 179.993607,s 2,t 43,e1 0.0,e2 0.0,e3 0.0,e4 0.0,e5 0.0,e6 0.0}
DECL FDAT FP177={TOOL_NO 1,BASE_NO 0,IPO_FRAME #BASE}
DECL PDAT PPDAT162={VEL 100.0,ACC 100.0,APO_DIST 100.0}
DECL E6POS XP178={x 66.1680298,y 1809.88098,z 2111.27588,a -92.4150772,b -2.27500892,c 179.992706,s 2,t 43,e1 0.0,e2 0.0,e3 0.0,e4 0.0,e5 0.0,e6 0.0}
DECL FDAT FP178={TOOL_NO 1,BASE_NO 0,IPO_FRAME #BASE}
DECL LDAT LCPDAT13={VEL 2.0,ACC 100.0,APO_DIST 100.0,APO_FAC 50.0}
DECL E6POS XP179={x 66.1682968,y 1809.88696,z 17.9583702,a -92.414917,b -2.27510691,c 179.992706,s 2,t 43,e1 0.0,e2 0.0,e3 0.0,e4 0.0,e5 0.0,e6 0.0}
DECL FDAT FP179={TOOL_NO 1,BASE_NO 0,IPO_FRAME #BASE}
DECL LDAT LCPDAT14={VEL 2.0,ACC 100.0,APO_DIST 100.0,APO_FAC 50.0}
DECL E6POS XP180={x 66.1656265,y 1809.89099,z 208.059204,a -92.2722168,b 0.153285295,c -88.8564987,s 2,t 35,e1 0.0,e2 0.0,e3 0.0,e4 0.0,e5 0.0,e6 0.0}
DECL FDAT FP180={TOOL_NO 1,BASE_NO 0,IPO_FRAME #BASE}
DECL PDAT PPDAT163={VEL 100.0,ACC 100.0,APO_DIST 100.0}
DECL E6POS XP181={x 1164.25403,y 1598.43298,z 835.157776,a -92.2723083,b 0.154096603,c -88.8562469,s 2,t 35,e1 0.0,e2 0.0,e3 0.0,e4 0.0,e5 0.0,e6 0.0}
DECL FDAT FP181={TOOL_NO 1,BASE_NO 0,IPO_FRAME #BASE}
DECL PDAT PPDAT164={VEL 100.0,ACC 100.0,APO_DIST 100.0}
DECL E6POS XP182={x -50.3950005,y -1685.53198,z 906.40033,a 88.0845718,b 24.8388309,c 178.952194,s 6,t 50,e1 0.0,e2 0.0,e3 0.0,e4 0.0,e5 0.0,e6 0.0}
DECL FDAT FP182={TOOL_NO 1,BASE_NO 0,IPO_FRAME #BASE}
DECL PDAT PPDAT165={VEL 100.0,ACC 100.0,APO_DIST 100.0}
DECL E6POS XP183={x -53.879921,y -1634.92102,z 98.8474274,a 61.5474701,b -2.54491711,c -178.662399,s 2,t 34,e1 0.0,e2 0.0,e3 0.0,e4 0.0,e5 0.0,e6 0.0}
DECL FDAT FP183={TOOL_NO 1,BASE_NO 0,IPO_FRAME #BASE}
DECL PDAT PPDAT166={VEL 100.0,ACC 100.0,APO_DIST 100.0}
DECL E6POS XP184={x -53.8190117,y -1918.15002,z 98.7891083,a 61.5484695,b -2.54965401,c -178.6604,s 2,t 34,e1 0.0,e2 0.0,e3 0.0,e4 0.0,e5 0.0,e6 0.0}
DECL FDAT FP184={TOOL_NO 1,BASE_NO 0,IPO_FRAME #BASE}
DECL PDAT PPDAT167={VEL 100.0,ACC 100.0,APO_DIST 100.0}
DECL E6POS XP185={x 1378.14697,y -1918.27502,z 98.8190308,a 61.5521584,b -2.55059099,c -178.662994,s 2,t 40,e1 0.0,e2 0.0,e3 0.0,e4 0.0,e5 0.0,e6 0.0}
DECL FDAT FP185={TOOL_NO 1,BASE_NO 0,IPO_FRAME #BASE}
DECL PDAT PPDAT168={VEL 100.0,ACC 100.0,APO_DIST 100.0}
DECL E6POS XP186={x 1378.57104,y -1041.46204,z 98.8533096,a 61.5378914,b -2.54018092,c -178.677399,s 2,t 42,e1 0.0,e2 0.0,e3 0.0,e4 0.0,e5 0.0,e6 0.0}
DECL FDAT FP186={TOOL_NO 1,BASE_NO 0,IPO_FRAME #BASE}
DECL PDAT PPDAT169={VEL 100.0,ACC 100.0,APO_DIST 100.0}
DECL E6POS XP187={x 2093.95801,y -993.6073,z 10.4236603,a 61.5541,b -2.55962396,c -178.712906,s 2,t 40,e1 0.0,e2 0.0,e3 0.0,e4 0.0,e5 0.0,e6 0.0}
DECL FDAT FP187={TOOL_NO 1,BASE_NO 0,IPO_FRAME #BASE}
DECL PDAT PPDAT170={VEL 100.0,ACC 100.0,APO_DIST 100.0}
DECL E6POS XP188={x 2093.52393,y 1121.59705,z 10.2355604,a 61.5238686,b -2.53641605,c -178.704605,s 2,t 41,e1 0.0,e2 0.0,e3 0.0,e4 0.0,e5 0.0,e6 0.0}
DECL FDAT FP188={TOOL_NO 1,BASE_NO 0,IPO_FRAME #BASE}
DECL PDAT PPDAT171={VEL 100.0,ACC 100.0,APO_DIST 100.0}
DECL E6POS XP189={x 1376.57104,y 1121.39502,z 2814.44995,a 118.588097,b 0.247895598,c 5.5229578,s 2,t 35,e1 0.0,e2 0.0,e3 0.0,e4 0.0,e5 0.0,e6 0.0}
DECL FDAT FP189={TOOL_NO 1,BASE_NO 0,IPO_FRAME #BASE}
DECL PDAT PPDAT172={VEL 100.0,ACC 100.0,APO_DIST 100.0}
DECL E6POS XP190={x -1618.38403,y 72.3351822,z 2194.88892,a 14.2926903,b 89.9889603,c -163.148102,s 2,t 2,e1 0.0,e2 0.0,e3 0.0,e4 0.0,e5 0.0,e6 0.0}
DECL FDAT FP190={TOOL_NO 1,BASE_NO 0,IPO_FRAME #BASE}
DECL PDAT PPDAT173={VEL 100.0,ACC 100.0,APO_DIST 100.0}
DECL E6POS XP191={x -2280.84497,y 112.090797,z 957.843384,a -3.68669891,b 85.4807968,c 178.121704,s 6,t 50,e1 0.0,e2 0.0,e3 0.0,e4 0.0,e5 0.0,e6 0.0}
DECL FDAT FP191={TOOL_NO 1,BASE_NO 0,IPO_FRAME #BASE}
DECL PDAT PPDAT174={VEL 100.0,ACC 100.0,APO_DIST 100.0}
DECL E6POS XP192={x -2280.85303,y 82.1072464,z 957.854004,a -3.68772292,b 85.4815292,c 178.120804,s 6,t 50,e1 0.0,e2 0.0,e3 0.0,e4 0.0,e5 0.0,e6 0.0}
DECL FDAT FP192={TOOL_NO 1,BASE_NO 0,IPO_FRAME #BASE}
DECL LDAT LCPDAT15={VEL 2.0,ACC 100.0,APO_DIST 100.0,APO_FAC 50.0}
DECL E6POS XP193={x -2281.0271,y -1477.06995,z 958.252014,a -3.91989994,b 85.4926529,c 177.8909,s 6,t 26,e1 0.0,e2 0.0,e3 0.0,e4 0.0,e5 0.0,e6 0.0}
DECL FDAT FP193={TOOL_NO 1,BASE_NO 0,IPO_FRAME #BASE}
DECL LDAT LCPDAT16={VEL 2.0,ACC 100.0,APO_DIST 100.0,APO_FAC 50.0}
DECL E6POS XP194={x -2280.42603,y -1445.21106,z 957.56073,a -3.45129108,b 85.4791031,c 178.322403,s 6,t 26,e1 0.0,e2 0.0,e3 0.0,e4 0.0,e5 0.0,e6 0.0}
DECL FDAT FP194={TOOL_NO 1,BASE_NO 0,IPO_FRAME #BASE}
DECL PDAT PPDAT175={VEL 100.0,ACC 100.0,APO_DIST 100.0}
DECL E6POS XP195={x -1512.81201,y -2268.37207,z 957.95459,a 151.033997,b 81.9740829,c -114.8097,s 6,t 50,e1 0.0,e2 0.0,e3 0.0,e4 0.0,e5 0.0,e6 0.0}
DECL FDAT FP195={TOOL_NO 1,BASE_NO 0,IPO_FRAME #BASE}
DECL PDAT PPDAT176={VEL 100.0,ACC 100.0,APO_DIST 100.0}
DECL E6POS XP196={x -1520.57104,y -2267.57788,z 957.12738,a 150.789902,b 82.012207,c -115.003601,s 6,t 50,e1 0.0,e2 0.0,e3 0.0,e4 0.0,e5 0.0,e6 0.0}
DECL FDAT FP196={TOOL_NO 1,BASE_NO 0,IPO_FRAME #BASE}
DECL LDAT LCPDAT17={VEL 2.0,ACC 100.0,APO_DIST 100.0,APO_FAC 50.0}
DECL E6POS XP197={x 1466.65002,y -2267.65894,z 957.347412,a 150.852203,b 82.0226974,c -114.9356,s 6,t 26,e1 0.0,e2 0.0,e3 0.0,e4 0.0,e5 0.0,e6 0.0}
DECL FDAT FP197={TOOL_NO 1,BASE_NO 0,IPO_FRAME #BASE}
DECL LDAT LCPDAT18={VEL 2.0,ACC 100.0,APO_DIST 100.0,APO_FAC 50.0}
DECL E6POS XP198={x 1585.62,y -2186.12988,z 957.366821,a 153.913605,b 82.0239868,c -114.934502,s 6,t 26,e1 0.0,e2 0.0,e3 0.0,e4 0.0,e5 0.0,e6 0.0}
DECL FDAT FP198={TOOL_NO 1,BASE_NO 0,IPO_FRAME #BASE}
DECL PDAT PPDAT177={VEL 100.0,ACC 100.0,APO_DIST 100.0}
DECL E6POS XP199={x 2261.15601,y -1500.12805,z 957.008911,a -117.474602,b 83.1847916,c -113.845802,s 6,t 50,e1 0.0,e2 0.0,e3 0.0,e4 0.0,e5 0.0,e6 0.0}
DECL FDAT FP199={TOOL_NO 1,BASE_NO 0,IPO_FRAME #BASE}
DECL PDAT PPDAT178={VEL 100.0,ACC 100.0,APO_DIST 100.0}
DECL E6POS XP200={x 2261.43506,y -1526.56702,z 957.461914,a -117.3601,b 83.1926727,c -113.758698,s 6,t 50,e1 0.0,e2 0.0,e3 0.0,e4 0.0,e5 0.0,e6 0.0}
DECL FDAT FP200={TOOL_NO 1,BASE_NO 0,IPO_FRAME #BASE}
DECL LDAT LCPDAT19={VEL 2.0,ACC 100.0,APO_DIST 100.0,APO_FAC 50.0}
DECL E6POS XP201={x 2261.61206,y 1485.48401,z 957.823486,a -117.379204,b 83.2153168,c -113.761597,s 6,t 27,e1 0.0,e2 0.0,e3 0.0,e4 0.0,e5 0.0,e6 0.0}
DECL FDAT FP201={TOOL_NO 1,BASE_NO 0,IPO_FRAME #BASE}
DECL LDAT LCPDAT20={VEL 2.0,ACC 100.0,APO_DIST 100.0,APO_FAC 50.0}
DECL E6POS XP202={x 2261.61206,y 1485.48401,z 957.823486,a -117.379204,b 83.2153168,c -113.761597,s 6,t 27,e1 0.0,e2 0.0,e3 0.0,e4 0.0,e5 0.0,e6 0.0}
DECL FDAT FP202={TOOL_NO 1,BASE_NO 0,IPO_FRAME #BASE}
DECL PDAT PPDAT179={VEL 100.0,ACC 100.0,APO_DIST 100.0}
DECL E6POS XP203={x 1508.68103,y 2260.26611,z 959.096375,a -12.3408699,b 74.4154587,c -98.824913,s 6,t 51,e1 0.0,e2 0.0,e3 0.0,e4 0.0,e5 0.0,e6 0.0}
DECL FDAT FP203={TOOL_NO 1,BASE_NO 0,IPO_FRAME #BASE}
DECL PDAT PPDAT180={VEL 100.0,ACC 100.0,APO_DIST 100.0}
DECL E6POS XP204={x 1500.12903,y 2259.99902,z 958.557617,a -12.4448795,b 74.400032,c -98.9111099,s 6,t 51,e1 0.0,e2 0.0,e3 0.0,e4 0.0,e5 0.0,e6 0.0}
DECL FDAT FP204={TOOL_NO 1,BASE_NO 0,IPO_FRAME #BASE}
DECL LDAT LCPDAT21={VEL 2.0,ACC 100.0,APO_DIST 100.0,APO_FAC 50.0}
DECL E6POS XP205={x -1494.52905,y 2260.177,z 958.841797,a -12.44804,b 74.4216614,c -98.8976212,s 6,t 27,e1 0.0,e2 0.0,e3 0.0,e4 0.0,e5 0.0,e6 0.0}
DECL FDAT FP205={TOOL_NO 1,BASE_NO 0,IPO_FRAME #BASE}
DECL LDAT LCPDAT22={VEL 2.0,ACC 100.0,APO_DIST 100.0,APO_FAC 50.0}
DECL E6POS XP206={x -1463.78699,y 2259.71094,z 958.278625,a -12.4290504,b 74.3730011,c -98.9252472,s 6,t 27,e1 0.0,e2 0.0,e3 0.0,e4 0.0,e5 0.0,e6 0.0}
DECL FDAT FP206={TOOL_NO 1,BASE_NO 0,IPO_FRAME #BASE}
DECL PDAT PPDAT181={VEL 100.0,ACC 100.0,APO_DIST 100.0}
DECL E6POS XP207={x -2228.61206,y 1569.95898,z 960.335876,a 75.4147415,b 74.3603897,c -99.2827606,s 6,t 51,e1 0.0,e2 0.0,e3 0.0,e4 0.0,e5 0.0,e6 0.0}
DECL FDAT FP207={TOOL_NO 1,BASE_NO 0,IPO_FRAME #BASE}
DECL PDAT PPDAT182={VEL 100.0,ACC 100.0,APO_DIST 100.0}
DECL E6POS XP208={x -2228.39502,y 1564.70996,z 960.163086,a 75.3728333,b 74.3557968,c -99.3130569,s 6,t 51,e1 0.0,e2 0.0,e3 0.0,e4 0.0,e5 0.0,e6 0.0}
DECL FDAT FP208={TOOL_NO 1,BASE_NO 0,IPO_FRAME #BASE}
DECL LDAT LCPDAT23={VEL 2.0,ACC 100.0,APO_DIST 100.0,APO_FAC 50.0}
DECL E6POS XP209={x -2228.6709,y -14.0335302,z 960.429871,a 73.8741913,b 74.0102234,c -103.358498,s 6,t 27,e1 0.0,e2 0.0,e3 0.0,e4 0.0,e5 0.0,e6 0.0}
DECL FDAT FP209={TOOL_NO 1,BASE_NO 0,IPO_FRAME #BASE}
DECL LDAT LCPDAT24={VEL 2.0,ACC 100.0,APO_DIST 100.0,APO_FAC 50.0}
DECL E6POS XP210={x -106.088997,y 7.34252977,z 3080.57495,a -3.96230412,b 3.45461392,c -0.000187530706,s 3,t 2,e1 0.0,e2 0.0,e3 0.0,e4 0.0,e5 0.0,e6 0.0}
DECL FDAT FP210={TOOL_NO 1,BASE_NO 0,IPO_FRAME #BASE}
DECL PDAT PPDAT183={VEL 100.0,ACC 100.0,APO_DIST 100.0}
DECL E6POS XP211={x 74.8183365,y 75.5588837,z 3080.57495,a -134.721207,b 3.45494008,c -0.000202915806,s 3,t 2,e1 0.0,e2 0.0,e3 0.0,e4 0.0,e5 0.0,e6 0.0}
DECL FDAT FP211={TOOL_NO 1,BASE_NO 0,IPO_FRAME #BASE}
DECL PDAT PPDAT184={VEL 100.0,ACC 100.0,APO_DIST 100.0}
DECL E6POS XP212={x -1395.09399,y -1406.82202,z 1806.45105,a -134.683502,b 21.4240704,c 0.0279728994,s 4,t 52,e1 0.0,e2 0.0,e3 0.0,e4 0.0,e5 0.0,e6 0.0}
DECL FDAT FP212={TOOL_NO 1,BASE_NO 0,IPO_FRAME #BASE}
DECL PDAT PPDAT185={VEL 100.0,ACC 100.0,APO_DIST 100.0}
DECL E6POS XP213={x -1898.59802,y -1815.88501,z 197.424103,a 43.5580482,b 64.7880173,c 179.849503,s 6,t 48,e1 0.0,e2 0.0,e3 0.0,e4 0.0,e5 0.0,e6 0.0}
DECL FDAT FP213={TOOL_NO 1,BASE_NO 0,IPO_FRAME #BASE}
DECL PDAT PPDAT186={VEL 100.0,ACC 100.0,APO_DIST 100.0}
DECL E6POS XP214={x 409.59671,y 391.750702,z 2943.38403,a -136.202698,b -14.1754799,c -0.0179368202,s 7,t 50,e1 0.0,e2 0.0,e3 0.0,e4 0.0,e5 0.0,e6 0.0}
DECL FDAT FP214={TOOL_NO 1,BASE_NO 0,IPO_FRAME #BASE}
DECL PDAT PPDAT187={VEL 100.0,ACC 100.0,APO_DIST 100.0}
DECL E6POS XP215={x 836.002197,y 799.578125,z 1226.40295,a 43.5912819,b -57.7241783,c -179.887604,s 5,t 54,e1 0.0,e2 0.0,e3 0.0,e4 0.0,e5 0.0,e6 0.0}
DECL FDAT FP215={TOOL_NO 1,BASE_NO 0,IPO_FRAME #BASE}
DECL PDAT PPDAT188={VEL 100.0,ACC 100.0,APO_DIST 100.0}
DECL E6POS XP216={x 1620.01697,y -0.00344053004,z 383.180298,a -162.175507,b 89.990448,c -162.175293,s 6,t 18,e1 0.0,e2 0.0,e3 0.0,e4 0.0,e5 0.0,e6 0.0}
DECL FDAT FP216={TOOL_NO 1,BASE_NO 0,IPO_FRAME #BASE}
DECL PDAT PPDAT189={VEL 100.0,ACC 100.0,APO_DIST 100.0}
DECL E6POS XP217={x 2520.31006,y -0.00478318101,z 383.71701,a 3.36560702,b 89.9933472,c 3.36560798,s 6,t 48,e1 0.0,e2 0.0,e3 0.0,e4 0.0,e5 0.0,e6 0.0}
DECL FDAT FP217={TOOL_NO 1,BASE_NO 0,IPO_FRAME #BASE}
DECL PDAT PPDAT190={VEL 100.0,ACC 100.0,APO_DIST 100.0}
DECL E6POS XP218={x 2452.35791,y -0.00208926806,z 922.55603,a 2.19463205,b 3.84193301,c 0.147564799,s 6,t 56,e1 0.0,e2 0.0,e3 0.0,e4 0.0,e5 0.0,e6 0.0}
DECL FDAT FP218={TOOL_NO 1,BASE_NO 0,IPO_FRAME #BASE}
DECL PDAT PPDAT191={VEL 100.0,ACC 100.0,APO_DIST 100.0}
DECL E6POS XP219={x 2180.87207,y 195.744095,z 2267.948,a 2.20100307,b 3.80813694,c 0.146124199,s 6,t 27,e1 0.0,e2 0.0,e3 0.0,e4 0.0,e5 0.0,e6 0.0}
DECL FDAT FP219={TOOL_NO 1,BASE_NO 0,IPO_FRAME #BASE}
DECL PDAT PPDAT192={VEL 100.0,ACC 100.0,APO_DIST 100.0}
DECL E6POS XP220={x 1621.55005,y -0.0137751503,z 1982.74194,a -90.1462784,b 61.6394081,c -90.1656723,s 6,t 18,e1 0.0,e2 0.0,e3 0.0,e4 0.0,e5 0.0,e6 0.0}
DECL FDAT FP220={TOOL_NO 1,BASE_NO 0,IPO_FRAME #BASE}
DECL PDAT PPDAT193={VEL 100.0,ACC 100.0,APO_DIST 100.0}
DECL E6POS XP221={x 2189.81299,y -0.0144306198,z 1989.422,a -90.1455536,b 61.6386909,c -90.1648788,s 6,t 26,e1 0.0,e2 0.0,e3 0.0,e4 0.0,e5 0.0,e6 0.0}
DECL FDAT FP221={TOOL_NO 1,BASE_NO 0,IPO_FRAME #BASE}
DECL PDAT PPDAT194={VEL 100.0,ACC 100.0,APO_DIST 100.0}
DECL E6POS XP222={x 2189.78809,y -30.3981895,z 1989.42102,a -90.1566391,b 61.6547699,c -90.1700287,s 6,t 18,e1 0.0,e2 0.0,e3 0.0,e4 0.0,e5 0.0,e6 0.0}
DECL FDAT FP222={TOOL_NO 1,BASE_NO 0,IPO_FRAME #BASE}
DECL LDAT LCPDAT25={VEL 2.0,ACC 100.0,APO_DIST 100.0,APO_FAC 50.0}
DECL E6POS XP223={x -753.667603,y 800.238525,z 2995.38794,a 98.8309784,b 18.5273991,c -16.0746307,s 2,t 35,e1 0.0,e2 0.0,e3 0.0,e4 0.0,e5 0.0,e6 0.0}
DECL FDAT FP223={TOOL_NO 1,BASE_NO 0,IPO_FRAME #BASE}
DECL PDAT PPDAT195={VEL 100.0,ACC 100.0,APO_DIST 100.0}
DECL E6POS XP224={x 663.358521,y 0.0215195697,z 2134.63892,a -28.3836594,b 2.49147606,c -1.35206699,s 6,t 18,e1 0.0,e2 0.0,e3 0.0,e4 0.0,e5 0.0,e6 0.0}
DECL FDAT FP224={TOOL_NO 1,BASE_NO 0,IPO_FRAME #BASE}
DECL PDAT PPDAT196={VEL 100.0,ACC 100.0,APO_DIST 100.0}
DECL E6POS XP225={x 650.045593,y 0.760956705,z 1594.96301,a 26.6041508,b -0.0802811012,c -179.858307,s 6,t 18,e1 0.0,e2 0.0,e3 0.0,e4 0.0,e5 0.0,e6 0.0}
DECL FDAT FP225={TOOL_NO 1,BASE_NO 0,IPO_FRAME #BASE}
DECL PDAT PPDAT197={VEL 100.0,ACC 100.0,APO_DIST 100.0}
DECL E6POS XP226={x -559.476624,y -575.614014,z 1642.28699,a -103.035301,b -30.4562607,c 163.0784,s 6,t 18,e1 0.0,e2 0.0,e3 0.0,e4 0.0,e5 0.0,e6 0.0}
DECL FDAT FP226={TOOL_NO 1,BASE_NO 0,IPO_FRAME #BASE}
DECL PDAT PPDAT198={VEL 100.0,ACC 100.0,APO_DIST 100.0}
DECL E6POS XP227={x -1471.64294,y -1495.86804,z 2072.63306,a 162.787903,b 54.5522194,c -56.7917786,s 6,t 26,e1 0.0,e2 0.0,e3 0.0,e4 0.0,e5 0.0,e6 0.0}
DECL FDAT FP227={TOOL_NO 1,BASE_NO 0,IPO_FRAME #BASE}
DECL PDAT PPDAT199={VEL 100.0,ACC 100.0,APO_DIST 100.0}
DECL E6POS XP228={x -188.994598,y -187.360504,z 2989.90405,a 94.6230698,b -2.32268,c -3.90681791,s 6,t 26,e1 0.0,e2 0.0,e3 0.0,e4 0.0,e5 0.0,e6 0.0}
DECL FDAT FP228={TOOL_NO 1,BASE_NO 0,IPO_FRAME #BASE}
DECL PDAT PPDAT200={VEL 100.0,ACC 100.0,APO_DIST 100.0}
DECL E6POS XP229={x 401.330688,y 414.865601,z 2966.29004,a 15.3127298,b 35.9474907,c -19.7910004,s 7,t 26,e1 0.0,e2 0.0,e3 0.0,e4 0.0,e5 0.0,e6 0.0}
DECL FDAT FP229={TOOL_NO 1,BASE_NO 0,IPO_FRAME #BASE}
DECL PDAT PPDAT201={VEL 100.0,ACC 100.0,APO_DIST 100.0}
DECL E6POS XP230={x 867.009583,y 885.993713,z 2081.49292,a -35.8031082,b 63.5691719,c -80.6354065,s 5,t 30,e1 0.0,e2 0.0,e3 0.0,e4 0.0,e5 0.0,e6 0.0}
DECL FDAT FP230={TOOL_NO 1,BASE_NO 0,IPO_FRAME #BASE}
DECL PDAT PPDAT202={VEL 100.0,ACC 100.0,APO_DIST 100.0}
DECL E6POS XP231={x 725.986023,y 728.050781,z 1739.06702,a 6.98750782,b 32.593399,c -21.0619297,s 1,t 14,e1 0.0,e2 0.0,e3 0.0,e4 0.0,e5 0.0,e6 0.0}
DECL FDAT FP231={TOOL_NO 1,BASE_NO 0,IPO_FRAME #BASE}
DECL PDAT PPDAT203={VEL 100.0,ACC 100.0,APO_DIST 100.0}
DECL E6POS XP232={x 663.275085,y 0.0233948994,z 3159.94702,a -28.3845596,b 2.49313498,c -1.35313201,s 6,t 18,e1 0.0,e2 0.0,e3 0.0,e4 0.0,e5 0.0,e6 0.0}
DECL FDAT FP232={TOOL_NO 1,BASE_NO 0,IPO_FRAME #BASE}
DECL PDAT PPDAT204={VEL 100.0,ACC 100.0,APO_DIST 100.0}
DECL E6POS XP233={x 549.336792,y 371.689697,z 3159.94897,a 5.69656897,b 2.49267912,c -1.35287094,s 6,t 19,e1 0.0,e2 0.0,e3 0.0,e4 0.0,e5 0.0,e6 0.0}
DECL FDAT FP233={TOOL_NO 1,BASE_NO 0,IPO_FRAME #BASE}
DECL PDAT PPDAT205={VEL 100.0,ACC 100.0,APO_DIST 100.0}
DECL E6POS XP234={x 1476.65002,y 1210.36096,z 2363.64697,a 124.277,b -63.6832008,c 95.7925262,s 2,t 43,e1 0.0,e2 0.0,e3 0.0,e4 0.0,e5 0.0,e6 0.0}
DECL FDAT FP234={TOOL_NO 1,BASE_NO 0,IPO_FRAME #BASE}
DECL PDAT PPDAT206={VEL 100.0,ACC 100.0,APO_DIST 100.0}
DECL E6POS XP235={x 1476.82898,y 1209.84302,z 2539.95605,a 110.101303,b -50.7062988,c 113.650703,s 2,t 35,e1 0.0,e2 0.0,e3 0.0,e4 0.0,e5 0.0,e6 0.0}
DECL FDAT FP235={TOOL_NO 1,BASE_NO 0,IPO_FRAME #BASE}
DECL PDAT PPDAT207={VEL 100.0,ACC 100.0,APO_DIST 100.0}
DECL E6POS XP236={x 1510.60803,y 1237.59802,z 2185.46191,a 88.7753906,b -38.0450287,c 143.610901,s 2,t 35,e1 0.0,e2 0.0,e3 0.0,e4 0.0,e5 0.0,e6 0.0}
DECL FDAT FP236={TOOL_NO 1,BASE_NO 0,IPO_FRAME #BASE}
DECL PDAT PPDAT208={VEL 100.0,ACC 100.0,APO_DIST 100.0}
DECL E6POS XP237={x -454.857086,y 399.073303,z 1349.83606,a 162.934006,b 1.64292598,c -175.6008,s 2,t 43,e1 0.0,e2 0.0,e3 0.0,e4 0.0,e5 0.0,e6 0.0}
DECL FDAT FP237={TOOL_NO 1,BASE_NO 0,IPO_FRAME #BASE}
DECL PDAT PPDAT209={VEL 100.0,ACC 100.0,APO_DIST 100.0}
DECL E6POS XP238={x -1625.79102,y 1526.93103,z 439.031097,a 37.4316292,b 61.17556,c -96.6106033,s 6,t 59,e1 0.0,e2 0.0,e3 0.0,e4 0.0,e5 0.0,e6 0.0}
DECL FDAT FP238={TOOL_NO 1,BASE_NO 0,IPO_FRAME #BASE}
DECL PDAT PPDAT210={VEL 100.0,ACC 100.0,APO_DIST 100.0}
DECL E6POS XP239={x 1365.37598,y -1763.65906,z 439.036285,a -151.617493,b 61.1756401,c -96.6095963,s 6,t 58,e1 0.0,e2 0.0,e3 0.0,e4 0.0,e5 0.0,e6 0.0}
DECL FDAT FP239={TOOL_NO 1,BASE_NO 0,IPO_FRAME #BASE}
DECL PDAT PPDAT211={VEL 100.0,ACC 100.0,APO_DIST 100.0}
DECL E6POS XP240={x -2224.96899,y -155.849197,z 439.041412,a 84.6441727,b 61.1754684,c -96.608551,s 6,t 58,e1 0.0,e2 0.0,e3 0.0,e4 0.0,e5 0.0,e6 0.0}
DECL FDAT FP240={TOOL_NO 1,BASE_NO 0,IPO_FRAME #BASE}
DECL PDAT PPDAT212={VEL 100.0,ACC 100.0,APO_DIST 100.0}
DECL E6POS XP241={x 1553.84497,y 463.647186,z 2193.52808,a -73.5295334,b 61.6397896,c -90.1635895,s 2,t 3,e1 0.0,e2 0.0,e3 0.0,e4 0.0,e5 0.0,e6 0.0}
DECL FDAT FP241={TOOL_NO 1,BASE_NO 0,IPO_FRAME #BASE}
DECL PDAT PPDAT213={VEL 100.0,ACC 100.0,APO_DIST 100.0}
DECL E6POS XP242={x 1204.86694,y 881.737183,z 2110.5,a -111.900398,b 17.1486092,c -108.859596,s 6,t 27,e1 0.0,e2 0.0,e3 0.0,e4 0.0,e5 0.0,e6 0.0}
DECL FDAT FP242={TOOL_NO 1,BASE_NO 0,IPO_FRAME #BASE}
DECL PDAT PPDAT214={VEL 100.0,ACC 100.0,APO_DIST 100.0}
DECL E6POS XP243={x 961.164612,y 970.943604,z 1924.5,a 19.6302795,b -1.863451,c -176.655807,s 6,t 27,e1 0.0,e2 0.0,e3 0.0,e4 0.0,e5 0.0,e6 0.0}
DECL FDAT FP243={TOOL_NO 1,BASE_NO 0,IPO_FRAME #BASE}
DECL PDAT PPDAT215={VEL 100.0,ACC 100.0,APO_DIST 100.0}
DECL E6POS XP244={x 957.184875,y 940.024719,z 2463.57593,a -164.947693,b 0.933255792,c -2.63765001,s 2,t 11,e1 0.0,e2 0.0,e3 0.0,e4 0.0,e5 0.0,e6 0.0}
DECL FDAT FP244={TOOL_NO 1,BASE_NO 0,IPO_FRAME #BASE}
DECL PDAT PPDAT216={VEL 100.0,ACC 100.0,APO_DIST 100.0}
DECL E6POS XP245={x 1472.78406,y 1216.17102,z 2403.35693,a 104.650002,b -57.9703598,c 121.3601,s 6,t 27,e1 0.0,e2 0.0,e3 0.0,e4 0.0,e5 0.0,e6 0.0}
DECL FDAT FP245={TOOL_NO 1,BASE_NO 0,IPO_FRAME #BASE}
DECL PDAT PPDAT217={VEL 100.0,ACC 100.0,APO_DIST 100.0}
DECL E6POS XP246={x 1452.70898,y 1202.66394,z 2529.72192,a 109.249702,b -58.6069984,c 116.633904,s 6,t 27,e1 0.0,e2 0.0,e3 0.0,e4 0.0,e5 0.0,e6 0.0}
DECL FDAT FP246={TOOL_NO 1,BASE_NO 0,IPO_FRAME #BASE}
DECL PDAT PPDAT218={VEL 100.0,ACC 100.0,APO_DIST 100.0}
DECL E6POS XP247={x -2362.65698,y 100.273903,z 489.134003,a 80.7296066,b 61.4606514,c -97.7149734,s 6,t 26,e1 0.0,e2 0.0,e3 0.0,e4 0.0,e5 0.0,e6 0.0}
DECL FDAT FP247={TOOL_NO 1,BASE_NO 0,IPO_FRAME #BASE}
DECL PDAT PPDAT219={VEL 100.0,ACC 100.0,APO_DIST 100.0}
DECL E6POS XP248={x 1646.96106,y -1696.97302,z 489.133209,a -142.696899,b 61.4606514,c -97.7148895,s 6,t 26,e1 0.0,e2 0.0,e3 0.0,e4 0.0,e5 0.0,e6 0.0}
DECL FDAT FP248={TOOL_NO 1,BASE_NO 0,IPO_FRAME #BASE}
DECL PDAT PPDAT220={VEL 100.0,ACC 100.0,APO_DIST 100.0}
DECL E6POS XP249={x 1775.23206,y 1562.28699,z 489.13089,a -55.4913788,b 61.4608688,c -97.715538,s 6,t 27,e1 0.0,e2 0.0,e3 0.0,e4 0.0,e5 0.0,e6 0.0}
DECL FDAT FP249={TOOL_NO 1,BASE_NO 0,IPO_FRAME #BASE}
DECL PDAT PPDAT221={VEL 100.0,ACC 100.0,APO_DIST 100.0}
DECL E6POS XP250={x -2364.68799,y 20.7261009,z 489.131012,a 82.6563568,b 61.4609985,c -97.7161636,s 6,t 27,e1 0.0,e2 0.0,e3 0.0,e4 0.0,e5 0.0,e6 0.0}
DECL FDAT FP250={TOOL_NO 1,BASE_NO 0,IPO_FRAME #BASE}
DECL PDAT PPDAT222={VEL 100.0,ACC 100.0,APO_DIST 100.0}
DECL E6POS XP251={x -1629.97998,y 914.77832,z 448.106415,a 18.2982502,b 50.0216599,c -139.934906,s 6,t 27,e1 0.0,e2 0.0,e3 0.0,e4 0.0,e5 0.0,e6 0.0}
DECL FDAT FP251={TOOL_NO 1,BASE_NO 0,IPO_FRAME #BASE}
DECL PDAT PPDAT223={VEL 100.0,ACC 100.0,APO_DIST 100.0}
DECL E6POS XP252={x -1629.97998,y 914.77832,z 448.106415,a 18.2982502,b 50.0216599,c -139.934906,s 6,t 27,e1 0.0,e2 0.0,e3 0.0,e4 0.0,e5 0.0,e6 0.0}
DECL FDAT FP252={TOOL_NO 1,BASE_NO 0,IPO_FRAME #BASE}
DECL LDAT LCPDAT26={VEL 2.0,ACC 100.0,APO_DIST 100.0,APO_FAC 50.0}
DECL E6POS XP253={x -878.409485,y 797.997192,z 466.174408,a 18.3273296,b 50.0215111,c -139.907196,s 6,t 19,e1 0.0,e2 0.0,e3 0.0,e4 0.0,e5 0.0,e6 0.0}
DECL FDAT FP253={TOOL_NO 1,BASE_NO 0,IPO_FRAME #BASE}
DECL LDAT LCPDAT27={VEL 2.0,ACC 100.0,APO_DIST 100.0,APO_FAC 50.0}
DECL E6POS XP254={x -943.911987,y 871.654175,z 466.179291,a 18.3276691,b 50.0208206,c -139.907303,s 6,t 19,e1 0.0,e2 0.0,e3 0.0,e4 0.0,e5 0.0,e6 0.0}
DECL FDAT FP254={TOOL_NO 1,BASE_NO 0,IPO_FRAME #BASE}
DECL LDAT LCPDAT28={VEL 2.0,ACC 100.0,APO_DIST 100.0,APO_FAC 50.0}
DECL E6POS XP255={x -1005.70203,y 883.442993,z 460.10321,a 18.3160801,b 50.0211105,c -139.917694,s 6,t 19,e1 0.0,e2 0.0,e3 0.0,e4 0.0,e5 0.0,e6 0.0}
DECL FDAT FP255={TOOL_NO 1,BASE_NO 0,IPO_FRAME #BASE}
DECL PDAT PPDAT224={VEL 100.0,ACC 100.0,APO_DIST 100.0}
DECL E6POS XP256={x -1005.68201,y 921.763916,z 460.1362,a 9.59784317,b 49.6940002,c -140.307297,s 6,t 19,e1 0.0,e2 0.0,e3 0.0,e4 0.0,e5 0.0,e6 0.0}
DECL FDAT FP256={TOOL_NO 1,BASE_NO 0,IPO_FRAME #BASE}
DECL LDAT LCPDAT29={VEL 2.0,ACC 100.0,APO_DIST 100.0,APO_FAC 50.0}
DECL E6POS XP257={x -1240.53796,y 961.909302,z 460.128204,a 9.59664917,b 49.6930618,c -140.308594,s 6,t 27,e1 0.0,e2 0.0,e3 0.0,e4 0.0,e5 0.0,e6 0.0}
DECL FDAT FP257={TOOL_NO 1,BASE_NO 0,IPO_FRAME #BASE}
DECL LDAT LCPDAT30={VEL 2.0,ACC 100.0,APO_DIST 100.0,APO_FAC 50.0}
DECL E6POS XP258={x -1607.47595,y 961.905823,z 445.295288,a 9.59617233,b 49.6926308,c -140.309204,s 6,t 27,e1 0.0,e2 0.0,e3 0.0,e4 0.0,e5 0.0,e6 0.0}
DECL FDAT FP258={TOOL_NO 1,BASE_NO 0,IPO_FRAME #BASE}
DECL LDAT LCPDAT31={VEL 2.0,ACC 100.0,APO_DIST 100.0,APO_FAC 50.0}
DECL E6POS XP259={x -1607.47095,y 961.903015,z 1323.21594,a 9.59615803,b 49.6923218,c -140.309296,s 6,t 27,e1 0.0,e2 0.0,e3 0.0,e4 0.0,e5 0.0,e6 0.0}
DECL FDAT FP259={TOOL_NO 1,BASE_NO 0,IPO_FRAME #BASE}
DECL PDAT PPDAT225={VEL 100.0,ACC 100.0,APO_DIST 100.0}
DECL E6POS XP260={x 1662.31995,y 863.640808,z 1323.203,a -112.055,b 49.6918297,c -140.310394,s 6,t 27,e1 0.0,e2 0.0,e3 0.0,e4 0.0,e5 0.0,e6 0.0}
DECL FDAT FP260={TOOL_NO 1,BASE_NO 0,IPO_FRAME #BASE}
DECL PDAT PPDAT226={VEL 100.0,ACC 100.0,APO_DIST 100.0}
DECL E6POS XP261={x 1710.79199,y 817.461426,z 1724.96594,a -70.9422836,b 61.8017807,c -97.8140411,s 6,t 19,e1 0.0,e2 0.0,e3 0.0,e4 0.0,e5 0.0,e6 0.0}
DECL FDAT FP261={TOOL_NO 1,BASE_NO 0,IPO_FRAME #BASE}
DECL PDAT PPDAT227={VEL 100.0,ACC 100.0,APO_DIST 100.0}
DECL E6POS XP262={x 1376.13306,y 653.010925,z 1352.11206,a -70.3238373,b 62.2379799,c -96.8638382,s 6,t 19,e1 0.0,e2 0.0,e3 0.0,e4 0.0,e5 0.0,e6 0.0}
DECL FDAT FP262={TOOL_NO 1,BASE_NO 0,IPO_FRAME #BASE}
DECL PDAT PPDAT228={VEL 100.0,ACC 100.0,APO_DIST 100.0}
DECL E6POS XP263={x 1342.31799,y 611.032227,z 1307.52502,a -101.925301,b 62.1607399,c -99.8238831,s 6,t 27,e1 0.0,e2 0.0,e3 0.0,e4 0.0,e5 0.0,e6 0.0}
DECL FDAT FP263={TOOL_NO 1,BASE_NO 0,IPO_FRAME #BASE}
DECL PDAT PPDAT229={VEL 100.0,ACC 100.0,APO_DIST 100.0}
DECL E6POS XP264={x 1342.31799,y 611.032227,z 1307.52502,a -101.925301,b 62.1607399,c -99.8238831,s 6,t 27,e1 0.0,e2 0.0,e3 0.0,e4 0.0,e5 0.0,e6 0.0}
DECL FDAT FP264={TOOL_NO 1,BASE_NO 0,IPO_FRAME #BASE}
DECL LDAT LCPDAT32={VEL 2.0,ACC 100.0,APO_DIST 100.0,APO_FAC 50.0}
DECL E6POS XP265={x 1410.18604,y 604.72522,z 1307.526,a -101.925301,b 62.1610794,c -99.823761,s 6,t 27,e1 0.0,e2 0.0,e3 0.0,e4 0.0,e5 0.0,e6 0.0}
DECL FDAT FP265={TOOL_NO 1,BASE_NO 0,IPO_FRAME #BASE}
DECL LDAT LCPDAT33={VEL 2.0,ACC 100.0,APO_DIST 100.0,APO_FAC 50.0}
DECL E6POS XP266={x 1420.974,y 683.199585,z 1307.53198,a -101.924599,b 62.1620407,c -99.8228226,s 6,t 27,e1 0.0,e2 0.0,e3 0.0,e4 0.0,e5 0.0,e6 0.0}
DECL FDAT FP266={TOOL_NO 1,BASE_NO 0,IPO_FRAME #BASE}
DECL LDAT LCPDAT34={VEL 2.0,ACC 100.0,APO_DIST 100.0,APO_FAC 50.0}
DECL E6POS XP267={x 1346.40503,y 687.035889,z 1307.52795,a -101.924698,b 62.1613693,c -99.8228912,s 6,t 27,e1 0.0,e2 0.0,e3 0.0,e4 0.0,e5 0.0,e6 0.0}
DECL FDAT FP267={TOOL_NO 1,BASE_NO 0,IPO_FRAME #BASE}
DECL LDAT LCPDAT35={VEL 2.0,ACC 100.0,APO_DIST 100.0,APO_FAC 50.0}
DECL E6POS XP268={x 1346.40405,y 612.114014,z 1307.526,a -101.924698,b 62.1611404,c -99.8228531,s 6,t 27,e1 0.0,e2 0.0,e3 0.0,e4 0.0,e5 0.0,e6 0.0}
DECL FDAT FP268={TOOL_NO 1,BASE_NO 0,IPO_FRAME #BASE}
DECL LDAT LCPDAT36={VEL 2.0,ACC 100.0,APO_DIST 100.0,APO_FAC 50.0}
DECL E6POS XP269={x 1422.97205,y 686.999695,z 1307.52502,a -101.925201,b 62.1613503,c -99.8232727,s 6,t 27,e1 0.0,e2 0.0,e3 0.0,e4 0.0,e5 0.0,e6 0.0}
DECL FDAT FP269={TOOL_NO 1,BASE_NO 0,IPO_FRAME #BASE}
DECL LDAT LCPDAT37={VEL 2.0,ACC 100.0,APO_DIST 100.0,APO_FAC 50.0}
DECL E6POS XP270={x 1442.81604,y 708.90863,z 1307.52002,a -63.6950188,b 61.9664993,c -101.202301,s 6,t 19,e1 0.0,e2 0.0,e3 0.0,e4 0.0,e5 0.0,e6 0.0}
DECL FDAT FP270={TOOL_NO 1,BASE_NO 0,IPO_FRAME #BASE}
DECL PDAT PPDAT230={VEL 100.0,ACC 100.0,APO_DIST 100.0}
DECL E6POS XP271={x 1744.08997,y 943.018372,z 1129.17896,a -108.8592,b 30.5565891,c -162.024307,s 6,t 51,e1 0.0,e2 0.0,e3 0.0,e4 0.0,e5 0.0,e6 0.0}
DECL FDAT FP271={TOOL_NO 1,BASE_NO 0,IPO_FRAME #BASE}
DECL PDAT PPDAT231={VEL 100.0,ACC 100.0,APO_DIST 100.0}
DECL E6POS XP272={x 1744.21301,y 942.866089,z 1129.448,a -108.859497,b 30.5723,c -162.015106,s 6,t 51,e1 0.0,e2 0.0,e3 0.0,e4 0.0,e5 0.0,e6 0.0}
DECL FDAT FP272={TOOL_NO 1,BASE_NO 0,IPO_FRAME #BASE}
DECL LDAT LCPDAT38={VEL 2.0,ACC 100.0,APO_DIST 100.0,APO_FAC 50.0}
DECL E6POS XP273={x 1773.54797,y 992.902588,z 274.158203,a -108.858498,b 30.5718803,c -162.015594,s 6,t 19,e1 0.0,e2 0.0,e3 0.0,e4 0.0,e5 0.0,e6 0.0}
DECL FDAT FP273={TOOL_NO 1,BASE_NO 0,IPO_FRAME #BASE}
DECL LDAT LCPDAT39={VEL 2.0,ACC 100.0,APO_DIST 100.0,APO_FAC 50.0}
DECL E6POS XP274={x 1766.36304,y 1026.98706,z 274.150909,a -108.859299,b 30.5713005,c -162.016403,s 6,t 19,e1 0.0,e2 0.0,e3 0.0,e4 0.0,e5 0.0,e6 0.0}
DECL FDAT FP274={TOOL_NO 1,BASE_NO 0,IPO_FRAME #BASE}
DECL PDAT PPDAT232={VEL 100.0,ACC 100.0,APO_DIST 100.0}
DECL E6POS XP275={x 1557.18701,y 1224.82202,z 139.208801,a -62.4971313,b 15.46667,c -176.223404,s 6,t 51,e1 0.0,e2 0.0,e3 0.0,e4 0.0,e5 0.0,e6 0.0}
DECL FDAT FP275={TOOL_NO 1,BASE_NO 0,IPO_FRAME #BASE}
DECL PDAT PPDAT233={VEL 100.0,ACC 100.0,APO_DIST 100.0}
DECL E6POS XP276={x 1507.14697,y 1213.04004,z 139.223801,a -62.8232193,b 16.0087204,c -175.917694,s 6,t 51,e1 0.0,e2 0.0,e3 0.0,e4 0.0,e5 0.0,e6 0.0}
DECL FDAT FP276={TOOL_NO 1,BASE_NO 0,IPO_FRAME #BASE}
DECL PDAT PPDAT234={VEL 100.0,ACC 100.0,APO_DIST 100.0}
DECL E6POS XP277={x 1507.14697,y 1213.04004,z 139.223801,a -62.8232193,b 16.0087204,c -175.917694,s 6,t 51,e1 0.0,e2 0.0,e3 0.0,e4 0.0,e5 0.0,e6 0.0}
DECL FDAT FP277={TOOL_NO 1,BASE_NO 0,IPO_FRAME #BASE}
DECL LDAT LCPDAT40={VEL 2.0,ACC 100.0,APO_DIST 100.0,APO_FAC 50.0}
DECL E6POS XP278={x 1270.82104,y 1214.95105,z 143.891602,a -62.8288994,b 16.0072803,c -175.920105,s 6,t 19,e1 0.0,e2 0.0,e3 0.0,e4 0.0,e5 0.0,e6 0.0}
DECL FDAT FP278={TOOL_NO 1,BASE_NO 0,IPO_FRAME #BASE}
DECL LDAT LCPDAT41={VEL 2.0,ACC 100.0,APO_DIST 100.0,APO_FAC 50.0}
DECL E6POS XP279={x 1349.58398,y 1154.25598,z 972.331787,a -62.8286591,b 16.00811,c -175.918396,s 6,t 51,e1 0.0,e2 0.0,e3 0.0,e4 0.0,e5 0.0,e6 0.0}
DECL FDAT FP279={TOOL_NO 1,BASE_NO 0,IPO_FRAME #BASE}
DECL LDAT LCPDAT42={VEL 2.0,ACC 100.0,APO_DIST 100.0,APO_FAC 50.0}
DECL E6POS XP280={x 1349.57397,y 1154.30005,z 972.338989,a 28.5184193,b 18.4561901,c -168.797501,s 6,t 51,e1 0.0,e2 0.0,e3 0.0,e4 0.0,e5 0.0,e6 0.0}
DECL FDAT FP280={TOOL_NO 1,BASE_NO 0,IPO_FRAME #BASE}
DECL PDAT PPDAT235={VEL 100.0,ACC 100.0,APO_DIST 100.0}
DECL E6POS XP281={x 904.932617,y 721.793518,z 1037.60999,a 27.4039307,b 20.1653996,c -168.7453,s 6,t 19,e1 0.0,e2 0.0,e3 0.0,e4 0.0,e5 0.0,e6 0.0}
DECL FDAT FP281={TOOL_NO 1,BASE_NO 0,IPO_FRAME #BASE}
DECL PDAT PPDAT236={VEL 100.0,ACC 100.0,APO_DIST 100.0}
DECL E6POS XP282={x 904.932617,y 721.793518,z 1037.60999,a 27.4039307,b 20.1653996,c -168.7453,s 6,t 19,e1 0.0,e2 0.0,e3 0.0,e4 0.0,e5 0.0,e6 0.0}
DECL FDAT FP282={TOOL_NO 1,BASE_NO 0,IPO_FRAME #BASE}
DECL LDAT LCPDAT43={VEL 2.0,ACC 100.0,APO_DIST 100.0,APO_FAC 50.0}
DECL E6POS XP283={x 900.566772,y 642.558594,z 1037.61401,a 27.4036293,b 20.1648808,c -168.745193,s 6,t 19,e1 0.0,e2 0.0,e3 0.0,e4 0.0,e5 0.0,e6 0.0}
DECL FDAT FP283={TOOL_NO 1,BASE_NO 0,IPO_FRAME #BASE}
DECL LDAT LCPDAT44={VEL 2.0,ACC 100.0,APO_DIST 100.0,APO_FAC 50.0}
DECL E6POS XP284={x 820.193604,y 785.482727,z 208.770996,a 27.4037704,b 20.1650009,c -168.745605,s 6,t 19,e1 0.0,e2 0.0,e3 0.0,e4 0.0,e5 0.0,e6 0.0}
DECL FDAT FP284={TOOL_NO 1,BASE_NO 0,IPO_FRAME #BASE}
DECL LDAT LCPDAT45={VEL 2.0,ACC 100.0,APO_DIST 100.0,APO_FAC 50.0}
DECL E6POS XP285={x 820.187988,y 785.479187,z 1095.64294,a 27.4040508,b 20.1648293,c -168.7453,s 6,t 19,e1 0.0,e2 0.0,e3 0.0,e4 0.0,e5 0.0,e6 0.0}
DECL FDAT FP285={TOOL_NO 1,BASE_NO 0,IPO_FRAME #BASE}
DECL LDAT LCPDAT46={VEL 2.0,ACC 100.0,APO_DIST 100.0,APO_FAC 50.0}
DECL E6POS XP286={x 605.956177,y 1.39932096,z 1348.30396,a -152.173401,b -2.84254694,c 177.348694,s 2,t 10,e1 0.0,e2 0.0,e3 0.0,e4 0.0,e5 0.0,e6 0.0}
DECL FDAT FP286={TOOL_NO 1,BASE_NO 0,IPO_FRAME #BASE}
DECL PDAT PPDAT237={VEL 100.0,ACC 100.0,APO_DIST 100.0}
DECL E6POS XP287={x 522.497375,y 1228.56604,z 2322.56201,a 89.9625626,b 54.9707909,c 30.8375397,s 6,t 27,e1 0.0,e2 0.0,e3 0.0,e4 0.0,e5 0.0,e6 0.0}
DECL FDAT FP287={TOOL_NO 1,BASE_NO 0,IPO_FRAME #BASE}
DECL PDAT PPDAT238={VEL 100.0,ACC 100.0,APO_DIST 100.0}
DECL E6POS XP288={x 517.190979,y 1224.27197,z 2319.15991,a 89.970787,b 54.9819603,c 30.8440609,s 6,t 27,e1 0.0,e2 0.0,e3 0.0,e4 0.0,e5 0.0,e6 0.0}
DECL FDAT FP288={TOOL_NO 1,BASE_NO 0,IPO_FRAME #BASE}
DECL LDAT LCPDAT47={VEL 2.0,ACC 100.0,APO_DIST 100.0,APO_FAC 50.0}
DECL E6POS XP289={x 537.510315,y 1224.26697,z 1542.70105,a 89.9699936,b 54.9825897,c 30.8436508,s 6,t 59,e1 0.0,e2 0.0,e3 0.0,e4 0.0,e5 0.0,e6 0.0}
DECL FDAT FP289={TOOL_NO 1,BASE_NO 0,IPO_FRAME #BASE}
DECL LDAT LCPDAT48={VEL 2.0,ACC 100.0,APO_DIST 100.0,APO_FAC 50.0}
DECL E6POS XP290={x 544.877014,y 1224.10706,z 1406.00696,a 89.9739075,b 54.9899712,c 30.8531094,s 6,t 59,e1 0.0,e2 0.0,e3 0.0,e4 0.0,e5 0.0,e6 0.0}
DECL FDAT FP290={TOOL_NO 1,BASE_NO 0,IPO_FRAME #BASE}
DECL LDAT LCPDAT49={VEL 2.0,ACC 100.0,APO_DIST 100.0,APO_FAC 50.0}
DECL E6POS XP291={x 544.877014,y 1224.10706,z 1406.00696,a 89.9739075,b 54.9899712,c 30.8531094,s 6,t 59,e1 0.0,e2 0.0,e3 0.0,e4 0.0,e5 0.0,e6 0.0}
DECL FDAT FP291={TOOL_NO 1,BASE_NO 0,IPO_FRAME #BASE}
DECL PDAT PPDAT239={VEL 100.0,ACC 100.0,APO_DIST 100.0}
DECL E6POS XP292={x 545.233887,y 1224.08105,z 1405.83606,a -92.5937805,b 75.7507324,c -150.962906,s 6,t 27,e1 0.0,e2 0.0,e3 0.0,e4 0.0,e5 0.0,e6 0.0}
DECL FDAT FP292={TOOL_NO 1,BASE_NO 0,IPO_FRAME #BASE}
DECL PDAT PPDAT240={VEL 100.0,ACC 100.0,APO_DIST 100.0}
DECL E6POS XP293={x 420.691498,y 990.554077,z 1194.67603,a -159.234695,b 2.50620699,c -176.5784,s 2,t 35,e1 0.0,e2 0.0,e3 0.0,e4 0.0,e5 0.0,e6 0.0}
DECL FDAT FP293={TOOL_NO 1,BASE_NO 0,IPO_FRAME #BASE}
DECL PDAT PPDAT241={VEL 100.0,ACC 100.0,APO_DIST 100.0}
DECL E6POS XP294={x 736.436401,y 1278.75696,z 1194.67004,a -158.782593,b 11.8334398,c -172.975693,s 2,t 35,e1 0.0,e2 0.0,e3 0.0,e4 0.0,e5 0.0,e6 0.0}
DECL FDAT FP294={TOOL_NO 1,BASE_NO 0,IPO_FRAME #BASE}
DECL PDAT PPDAT242={VEL 100.0,ACC 100.0,APO_DIST 100.0}
DECL E6POS XP295={x 720.559814,y 1295.21106,z 1263.12305,a 176.317795,b 11.7334204,c -173.018799,s 2,t 35,e1 0.0,e2 0.0,e3 0.0,e4 0.0,e5 0.0,e6 0.0}
DECL FDAT FP295={TOOL_NO 1,BASE_NO 0,IPO_FRAME #BASE}
DECL PDAT PPDAT243={VEL 100.0,ACC 100.0,APO_DIST 100.0}
DECL E6POS XP296={x 720.559814,y 1295.21106,z 1263.12305,a 176.317795,b 11.7334204,c -173.018799,s 2,t 35,e1 0.0,e2 0.0,e3 0.0,e4 0.0,e5 0.0,e6 0.0}
DECL FDAT FP296={TOOL_NO 1,BASE_NO 0,IPO_FRAME #BASE}
DECL LDAT LCPDAT50={VEL 2.0,ACC 100.0,APO_DIST 100.0,APO_FAC 50.0}
DECL E6POS XP297={x 745.339478,y 1291.45605,z 156.150299,a 176.324707,b 11.7303801,c -173.018295,s 2,t 35,e1 0.0,e2 0.0,e3 0.0,e4 0.0,e5 0.0,e6 0.0}
DECL FDAT FP297={TOOL_NO 1,BASE_NO 0,IPO_FRAME #BASE}
DECL LDAT LCPDAT51={VEL 2.0,ACC 100.0,APO_DIST 100.0,APO_FAC 50.0}
DECL E6POS XP298={x 745.06012,y 1291.58801,z 156.310898,a 178.529495,b 16.9130592,c -172.513397,s 2,t 35,e1 0.0,e2 0.0,e3 0.0,e4 0.0,e5 0.0,e6 0.0}
DECL FDAT FP298={TOOL_NO 1,BASE_NO 0,IPO_FRAME #BASE}
DECL PDAT PPDAT244={VEL 100.0,ACC 100.0,APO_DIST 100.0}
DECL E6POS XP299={x 1122.24597,y 900.437073,z 2169.23511,a 160.764206,b 16.9136505,c -172.514297,s 2,t 35,e1 0.0,e2 0.0,e3 0.0,e4 0.0,e5 0.0,e6 0.0}
DECL FDAT FP299={TOOL_NO 1,BASE_NO 0,IPO_FRAME #BASE}
DECL PDAT PPDAT245={VEL 100.0,ACC 100.0,APO_DIST 100.0}
DECL E6POS XP300={x 1731.81006,y 80.0569611,z 1291.86401,a -94.7680969,b 61.5187111,c -95.4101028,s 6,t 27,e1 0.0,e2 0.0,e3 0.0,e4 0.0,e5 0.0,e6 0.0}
DECL FDAT FP300={TOOL_NO 1,BASE_NO 0,IPO_FRAME #BASE}
DECL PDAT PPDAT246={VEL 100.0,ACC 100.0,APO_DIST 100.0}
DECL E6POS XP301={x 1731.81006,y 80.0569611,z 1291.86401,a -94.7680969,b 61.5187111,c -95.4101028,s 6,t 27,e1 0.0,e2 0.0,e3 0.0,e4 0.0,e5 0.0,e6 0.0}
DECL FDAT FP301={TOOL_NO 1,BASE_NO 0,IPO_FRAME #BASE}
DECL LDAT LCPDAT52={VEL 2.0,ACC 100.0,APO_DIST 100.0,APO_FAC 50.0}
DECL E6POS XP302={x 1722.30505,y 71.4861679,z 1291.86206,a -94.7692032,b 61.5182114,c -95.4110565,s 6,t 27,e1 0.0,e2 0.0,e3 0.0,e4 0.0,e5 0.0,e6 0.0}
DECL FDAT FP302={TOOL_NO 1,BASE_NO 0,IPO_FRAME #BASE}
DECL LDAT LCPDAT53={VEL 2.0,ACC 100.0,APO_DIST 100.0,APO_FAC 50.0}
DECL E6POS XP303={x 1741.052,y 71.4911499,z 1291.87903,a -94.7666931,b 61.5182991,c -95.4080963,s 6,t 27,e1 0.0,e2 0.0,e3 0.0,e4 0.0,e5 0.0,e6 0.0}
DECL FDAT FP303={TOOL_NO 1,BASE_NO 0,IPO_FRAME #BASE}
DECL LDAT LCPDAT54={VEL 2.0,ACC 100.0,APO_DIST 100.0,APO_FAC 50.0}
DECL E6POS XP304={x 1741.05396,y 89.2674866,z 1291.88098,a -94.7663422,b 61.5180283,c -95.4075928,s 6,t 27,e1 0.0,e2 0.0,e3 0.0,e4 0.0,e5 0.0,e6 0.0}
DECL FDAT FP304={TOOL_NO 1,BASE_NO 0,IPO_FRAME #BASE}
DECL LDAT LCPDAT55={VEL 2.0,ACC 100.0,APO_DIST 100.0,APO_FAC 50.0}
DECL E6POS XP305={x 1721.73096,y 89.2692795,z 1291.85596,a -94.7688293,b 61.5168915,c -95.4108734,s 6,t 27,e1 0.0,e2 0.0,e3 0.0,e4 0.0,e5 0.0,e6 0.0}
DECL FDAT FP305={TOOL_NO 1,BASE_NO 0,IPO_FRAME #BASE}
DECL LDAT LCPDAT56={VEL 2.0,ACC 100.0,APO_DIST 100.0,APO_FAC 50.0}
DECL E6POS XP306={x 1721.72498,y 73.4645767,z 1291.84802,a -94.7700424,b 61.5173111,c -95.4122162,s 6,t 27,e1 0.0,e2 0.0,e3 0.0,e4 0.0,e5 0.0,e6 0.0}
DECL FDAT FP306={TOOL_NO 1,BASE_NO 0,IPO_FRAME #BASE}
DECL LDAT LCPDAT57={VEL 2.0,ACC 100.0,APO_DIST 100.0,APO_FAC 50.0}
DECL E6POS XP307={x 1721.72498,y 73.4645767,z 1291.84802,a -94.7700424,b 61.5173111,c -95.4122162,s 6,t 27,e1 0.0,e2 0.0,e3 0.0,e4 0.0,e5 0.0,e6 0.0}
DECL FDAT FP307={TOOL_NO 1,BASE_NO 0,IPO_FRAME #BASE}
DECL PDAT PPDAT247={VEL 100.0,ACC 100.0,APO_DIST 100.0}
DECL E6POS XP308={x 1783.68298,y -186.734802,z 1291.88,a -94.7656021,b 61.5183411,c -95.4075928,s 6,t 18,e1 0.0,e2 0.0,e3 0.0,e4 0.0,e5 0.0,e6 0.0}
DECL FDAT FP308={TOOL_NO 1,BASE_NO 0,IPO_FRAME #BASE}
DECL PDAT PPDAT248={VEL 100.0,ACC 100.0,APO_DIST 100.0}
DECL E6POS XP309={x 1785.85803,y -186.737595,z 1108.54797,a -94.7637177,b 61.5178108,c -95.4055862,s 6,t 18,e1 0.0,e2 0.0,e3 0.0,e4 0.0,e5 0.0,e6 0.0}
DECL FDAT FP309={TOOL_NO 1,BASE_NO 0,IPO_FRAME #BASE}
DECL PDAT PPDAT249={VEL 100.0,ACC 100.0,APO_DIST 100.0}
DECL E6POS XP310={x 1785.85803,y -186.737595,z 1108.54797,a -94.7637177,b 61.5178108,c -95.4055862,s 6,t 18,e1 0.0,e2 0.0,e3 0.0,e4 0.0,e5 0.0,e6 0.0}
DECL FDAT FP310={TOOL_NO 1,BASE_NO 0,IPO_FRAME #BASE}
DECL LDAT LCPDAT58={VEL 2.0,ACC 100.0,APO_DIST 100.0,APO_FAC 50.0}
DECL E6POS XP311={x 1946.21399,y -189.657196,z 1106.25696,a -94.7638931,b 61.5176582,c -95.4065323,s 6,t 18,e1 0.0,e2 0.0,e3 0.0,e4 0.0,e5 0.0,e6 0.0}
DECL FDAT FP311={TOOL_NO 1,BASE_NO 0,IPO_FRAME #BASE}
DECL LDAT LCPDAT59={VEL 2.0,ACC 100.0,APO_DIST 100.0,APO_FAC 50.0}
DECL E6POS XP312={x 1958.13904,y 335.881104,z 1106.26697,a -94.7629471,b 61.5179214,c -95.4053116,s 6,t 27,e1 0.0,e2 0.0,e3 0.0,e4 0.0,e5 0.0,e6 0.0}
DECL FDAT FP312={TOOL_NO 1,BASE_NO 0,IPO_FRAME #BASE}
DECL LDAT LCPDAT60={VEL 2.0,ACC 100.0,APO_DIST 100.0,APO_FAC 50.0}
DECL E6POS XP313={x 1800.09302,y 338.830292,z 1108.89697,a -94.7643967,b 61.5165787,c -95.4071198,s 6,t 27,e1 0.0,e2 0.0,e3 0.0,e4 0.0,e5 0.0,e6 0.0}
DECL FDAT FP313={TOOL_NO 1,BASE_NO 0,IPO_FRAME #BASE}
DECL LDAT LCPDAT61={VEL 2.0,ACC 100.0,APO_DIST 100.0,APO_FAC 50.0}
DECL E6POS XP314={x 1800.08899,y 269.132599,z 1110.44995,a -94.7659531,b 61.5165405,c -95.4086914,s 6,t 27,e1 0.0,e2 0.0,e3 0.0,e4 0.0,e5 0.0,e6 0.0}
DECL FDAT FP314={TOOL_NO 1,BASE_NO 0,IPO_FRAME #BASE}
DECL LDAT LCPDAT62={VEL 2.0,ACC 100.0,APO_DIST 100.0,APO_FAC 50.0}
DECL E6POS XP315={x 1768.38196,y 238.385101,z 1146.63501,a -94.7684326,b 61.5153389,c -95.4104614,s 6,t 27,e1 0.0,e2 0.0,e3 0.0,e4 0.0,e5 0.0,e6 0.0}
DECL FDAT FP315={TOOL_NO 1,BASE_NO 0,IPO_FRAME #BASE}
DECL PDAT PPDAT250={VEL 100.0,ACC 100.0,APO_DIST 100.0}
DECL E6POS XP316={x 1796.06897,y 226.3759,z 1125.21802,a -94.7700729,b 61.5161018,c -95.4109268,s 6,t 27,e1 0.0,e2 0.0,e3 0.0,e4 0.0,e5 0.0,e6 0.0}
DECL FDAT FP316={TOOL_NO 1,BASE_NO 0,IPO_FRAME #BASE}
DECL PDAT PPDAT251={VEL 100.0,ACC 100.0,APO_DIST 100.0}
DECL E6POS XP317={x 1796.08997,y 226.376999,z 1110.08301,a -94.7679672,b 61.5146294,c -95.4081497,s 6,t 27,e1 0.0,e2 0.0,e3 0.0,e4 0.0,e5 0.0,e6 0.0}
DECL FDAT FP317={TOOL_NO 1,BASE_NO 0,IPO_FRAME #BASE}
DECL PDAT PPDAT252={VEL 100.0,ACC 100.0,APO_DIST 100.0}
DECL E6POS XP318={x 1796.08997,y 226.376999,z 1110.08301,a -94.7679672,b 61.5146294,c -95.4081497,s 6,t 27,e1 0.0,e2 0.0,e3 0.0,e4 0.0,e5 0.0,e6 0.0}
DECL FDAT FP318={TOOL_NO 1,BASE_NO 0,IPO_FRAME #BASE}
DECL LDAT LCPDAT63={VEL 2.0,ACC 100.0,APO_DIST 100.0,APO_FAC 50.0}
DECL E6POS XP319={x 1796.08997,y 147.872299,z 1110.08203,a -94.7680969,b 61.514389,c -95.4083328,s 6,t 27,e1 0.0,e2 0.0,e3 0.0,e4 0.0,e5 0.0,e6 0.0}
DECL FDAT FP319={TOOL_NO 1,BASE_NO 0,IPO_FRAME #BASE}
DECL LDAT LCPDAT64={VEL 2.0,ACC 100.0,APO_DIST 100.0,APO_FAC 50.0}
DECL E6POS XP320={x 1796.08301,y 147.870697,z 1299.44104,a -94.7688065,b 61.5143509,c -95.4089127,s 6,t 27,e1 0.0,e2 0.0,e3 0.0,e4 0.0,e5 0.0,e6 0.0}
DECL FDAT FP320={TOOL_NO 1,BASE_NO 0,IPO_FRAME #BASE}
DECL PDAT PPDAT253={VEL 100.0,ACC 100.0,APO_DIST 100.0}
DECL E6POS XP321={x 1461.16199,y 173.845398,z 1194.59705,a 31.6446705,b 9.86890984,c -167.364502,s 2,t 11,e1 0.0,e2 0.0,e3 0.0,e4 0.0,e5 0.0,e6 0.0}
DECL FDAT FP321={TOOL_NO 1,BASE_NO 0,IPO_FRAME #BASE}
DECL PDAT PPDAT254={VEL 100.0,ACC 100.0,APO_DIST 100.0}
DECL E6POS XP322={x 1222.74695,y 49.3981781,z 910.479675,a 31.6415901,b 9.86982822,c -167.364502,s 2,t 11,e1 0.0,e2 0.0,e3 0.0,e4 0.0,e5 0.0,e6 0.0}
DECL FDAT FP322={TOOL_NO 1,BASE_NO 0,IPO_FRAME #BASE}
DECL PDAT PPDAT255={VEL 100.0,ACC 100.0,APO_DIST 100.0}
DECL E6POS XP323={x 1257.00598,y -65.8414688,z 910.487488,a 38.7779007,b 8.21354103,c -166.241898,s 2,t 10,e1 0.0,e2 0.0,e3 0.0,e4 0.0,e5 0.0,e6 0.0}
DECL FDAT FP323={TOOL_NO 1,BASE_NO 0,IPO_FRAME #BASE}
DECL PDAT PPDAT256={VEL 100.0,ACC 100.0,APO_DIST 100.0}
DECL E6POS XP324={x 1285.68701,y -35.5453987,z 718.87793,a 38.7752304,b 8.21167374,c -166.242996,s 2,t 10,e1 0.0,e2 0.0,e3 0.0,e4 0.0,e5 0.0,e6 0.0}
DECL FDAT FP324={TOOL_NO 1,BASE_NO 0,IPO_FRAME #BASE}
DECL PDAT PPDAT257={VEL 100.0,ACC 100.0,APO_DIST 100.0}
DECL E6POS XP325={x 1285.68701,y -35.5453987,z 718.87793,a 38.7752304,b 8.21167374,c -166.242996,s 2,t 10,e1 0.0,e2 0.0,e3 0.0,e4 0.0,e5 0.0,e6 0.0}
DECL FDAT FP325={TOOL_NO 1,BASE_NO 0,IPO_FRAME #BASE}
DECL LDAT LCPDAT65={VEL 2.0,ACC 100.0,APO_DIST 100.0,APO_FAC 50.0}
DECL E6POS XP326={x 1281.54004,y -277.93631,z 718.868225,a 38.7764816,b 8.21188068,c -166.244797,s 2,t 10,e1 0.0,e2 0.0,e3 0.0,e4 0.0,e5 0.0,e6 0.0}
DECL FDAT FP326={TOOL_NO 1,BASE_NO 0,IPO_FRAME #BASE}
DECL LDAT LCPDAT66={VEL 2.0,ACC 100.0,APO_DIST 100.0,APO_FAC 50.0}
DECL E6POS XP327={x 1281.54004,y -277.93631,z 718.868225,a 38.7764816,b 8.21188068,c -166.244797,s 2,t 10,e1 0.0,e2 0.0,e3 0.0,e4 0.0,e5 0.0,e6 0.0}
DECL FDAT FP327={TOOL_NO 1,BASE_NO 0,IPO_FRAME #BASE}
DECL PDAT PPDAT258={VEL 100.0,ACC 100.0,APO_DIST 100.0}
DECL E6POS XP328={x 1565.76099,y -604.174072,z 813.528503,a 90.0067596,b 13.3292799,c -154.882507,s 2,t 2,e1 0.0,e2 0.0,e3 0.0,e4 0.0,e5 0.0,e6 0.0}
DECL FDAT FP328={TOOL_NO 1,BASE_NO 0,IPO_FRAME #BASE}
DECL PDAT PPDAT259={VEL 100.0,ACC 100.0,APO_DIST 100.0}
DECL E6POS XP329={x 1565.76099,y -604.174072,z 813.528503,a 90.0067596,b 13.3292799,c -154.882507,s 2,t 2,e1 0.0,e2 0.0,e3 0.0,e4 0.0,e5 0.0,e6 0.0}
DECL FDAT FP329={TOOL_NO 1,BASE_NO 0,IPO_FRAME #BASE}
DECL LDAT LCPDAT67={VEL 2.0,ACC 100.0,APO_DIST 100.0,APO_FAC 50.0}
DECL E6POS XP330={x 1726.61499,y -607.721619,z 811.593811,a 90.0031967,b 13.33426,c -154.889297,s 2,t 2,e1 0.0,e2 0.0,e3 0.0,e4 0.0,e5 0.0,e6 0.0}
DECL FDAT FP330={TOOL_NO 1,BASE_NO 0,IPO_FRAME #BASE}
DECL LDAT LCPDAT68={VEL 2.0,ACC 100.0,APO_DIST 100.0,APO_FAC 50.0}
DECL E6POS XP331={x 1726.60706,y -609.788574,z 810.068787,a 90.0037766,b 13.3345804,c -154.889297,s 2,t 2,e1 0.0,e2 0.0,e3 0.0,e4 0.0,e5 0.0,e6 0.0}
DECL FDAT FP331={TOOL_NO 1,BASE_NO 0,IPO_FRAME #BASE}
DECL PDAT PPDAT260={VEL 100.0,ACC 100.0,APO_DIST 100.0}
DECL E6POS XP332={x 1726.60706,y -609.788574,z 810.068787,a 90.0037766,b 13.3345804,c -154.889297,s 2,t 2,e1 0.0,e2 0.0,e3 0.0,e4 0.0,e5 0.0,e6 0.0}
DECL FDAT FP332={TOOL_NO 1,BASE_NO 0,IPO_FRAME #BASE}
DECL LDAT LCPDAT69={VEL 2.0,ACC 100.0,APO_DIST 100.0,APO_FAC 50.0}
DECL E6POS XP333={x 1724.28699,y -609.76178,z 664.170288,a 90.0053864,b 13.3331203,c -154.888107,s 2,t 2,e1 0.0,e2 0.0,e3 0.0,e4 0.0,e5 0.0,e6 0.0}
DECL FDAT FP333={TOOL_NO 1,BASE_NO 0,IPO_FRAME #BASE}
DECL LDAT LCPDAT70={VEL 2.0,ACC 100.0,APO_DIST 100.0,APO_FAC 50.0}
DECL E6POS XP334={x 1768.86401,y -610.062012,z 659.68042,a 89.9978409,b 13.3387403,c -154.891098,s 2,t 2,e1 0.0,e2 0.0,e3 0.0,e4 0.0,e5 0.0,e6 0.0}
DECL FDAT FP334={TOOL_NO 1,BASE_NO 0,IPO_FRAME #BASE}
DECL LDAT LCPDAT71={VEL 2.0,ACC 100.0,APO_DIST 100.0,APO_FAC 50.0}
DECL E6POS XP335={x 1768.854,y -649.731689,z 645.690674,a 89.9978638,b 13.3380003,c -154.890198,s 2,t 2,e1 0.0,e2 0.0,e3 0.0,e4 0.0,e5 0.0,e6 0.0}
DECL FDAT FP335={TOOL_NO 1,BASE_NO 0,IPO_FRAME #BASE}
DECL LDAT LCPDAT72={VEL 2.0,ACC 100.0,APO_DIST 100.0,APO_FAC 50.0}
DECL E6POS XP336={x 1789.74097,y -633.359924,z 645.91217,a 89.9806671,b 13.3516998,c -154.904205,s 2,t 2,e1 0.0,e2 0.0,e3 0.0,e4 0.0,e5 0.0,e6 0.0}
DECL FDAT FP336={TOOL_NO 1,BASE_NO 0,IPO_FRAME #BASE}
DECL LDAT LCPDAT73={VEL 2.0,ACC 100.0,APO_DIST 100.0,APO_FAC 50.0}
DECL E6POS XP337={x 1787.53198,y -807.327515,z 645.886292,a 89.9829865,b 13.3503399,c -154.901794,s 2,t 2,e1 0.0,e2 0.0,e3 0.0,e4 0.0,e5 0.0,e6 0.0}
DECL FDAT FP337={TOOL_NO 1,BASE_NO 0,IPO_FRAME #BASE}
DECL LDAT LCPDAT74={VEL 2.0,ACC 100.0,APO_DIST 100.0,APO_FAC 50.0}
DECL E6POS XP338={x 1783.01001,y -818.505676,z 645.867126,a 89.9842682,b 13.3486996,c -154.899704,s 2,t 2,e1 0.0,e2 0.0,e3 0.0,e4 0.0,e5 0.0,e6 0.0}
DECL E6POS XP339={x 1753.74695,y -834.422729,z 645.693787,a 90.0043564,b 13.3366604,c -154.885895,s 2,t 2,e1 0.0,e2 0.0,e3 0.0,e4 0.0,e5 0.0,e6 0.0}
DECL FDAT FP339={TOOL_NO 1,BASE_NO 0,IPO_FRAME #BASE}
DECL LDAT LCPDAT75={VEL 2.0,ACC 100.0,APO_DIST 100.0,APO_FAC 50.0}
DECL E6POS XP340={x 1753.74695,y -834.422729,z 645.693787,a 90.0043564,b 13.3366604,c -154.885895,s 2,t 2,e1 0.0,e2 0.0,e3 0.0,e4 0.0,e5 0.0,e6 0.0}
DECL FDAT FP340={TOOL_NO 1,BASE_NO 0,IPO_FRAME #BASE}
DECL LDAT LCPDAT76={VEL 2.0,ACC 100.0,APO_DIST 100.0,APO_FAC 50.0}
DECL E6POS XP341={x 1526.76294,y -830.151306,z 645.672607,a 90.0084305,b 13.3341398,c -154.883804,s 2,t 2,e1 0.0,e2 0.0,e3 0.0,e4 0.0,e5 0.0,e6 0.0}
DECL FDAT FP341={TOOL_NO 1,BASE_NO 0,IPO_FRAME #BASE}
DECL LDAT LCPDAT77={VEL 2.0,ACC 100.0,APO_DIST 100.0,APO_FAC 50.0}
DECL E6POS XP342={x 1526.76099,y -830.153687,z 1522.24597,a 90.0081635,b 13.33395,c -154.883698,s 2,t 2,e1 0.0,e2 0.0,e3 0.0,e4 0.0,e5 0.0,e6 0.0}
DECL FDAT FP342={TOOL_NO 1,BASE_NO 0,IPO_FRAME #BASE}
DECL PDAT PPDAT261={VEL 100.0,ACC 100.0,APO_DIST 100.0}
DECL E6POS XP343={x 1526.75195,y -830.150024,z 645.669495,a 90.0084534,b 13.3338804,c -154.883194,s 2,t 2,e1 0.0,e2 0.0,e3 0.0,e4 0.0,e5 0.0,e6 0.0}
DECL FDAT FP343={TOOL_NO 1,BASE_NO 0,IPO_FRAME #BASE}
DECL LDAT LCPDAT78={VEL 2.0,ACC 100.0,APO_DIST 100.0,APO_FAC 50.0}
DECL E6POS XP344={x 1500.22302,y -821.283081,z 645.671082,a 90.0102005,b 13.3332195,c -154.882202,s 2,t 2,e1 0.0,e2 0.0,e3 0.0,e4 0.0,e5 0.0,e6 0.0}
DECL E6POS XP345={x 1486.71106,y -794.679993,z 645.669617,a 90.0109482,b 13.33284,c -154.880997,s 2,t 2,e1 0.0,e2 0.0,e3 0.0,e4 0.0,e5 0.0,e6 0.0}
DECL FDAT FP345={TOOL_NO 1,BASE_NO 0,IPO_FRAME #BASE}
DECL LDAT LCPDAT79={VEL 2.0,ACC 100.0,APO_DIST 100.0,APO_FAC 50.0}
DECL E6POS XP346={x 1486.71106,y -794.679993,z 645.669617,a 90.0109482,b 13.33284,c -154.880997,s 2,t 2,e1 0.0,e2 0.0,e3 0.0,e4 0.0,e5 0.0,e6 0.0}
DECL FDAT FP346={TOOL_NO 1,BASE_NO 0,IPO_FRAME #BASE}
DECL LDAT LCPDAT80={VEL 2.0,ACC 100.0,APO_DIST 100.0,APO_FAC 50.0}
DECL E6POS XP347={x 1490.60999,y -629.272888,z 645.677185,a 90.0103989,b 13.3333197,c -154.881805,s 2,t 2,e1 0.0,e2 0.0,e3 0.0,e4 0.0,e5 0.0,e6 0.0}
DECL FDAT FP347={TOOL_NO 1,BASE_NO 0,IPO_FRAME #BASE}
DECL LDAT LCPDAT81={VEL 2.0,ACC 100.0,APO_DIST 100.0,APO_FAC 50.0}
DECL E6POS XP348={x 1490.60999,y -629.272888,z 645.677185,a 90.0103989,b 13.3333197,c -154.881805,s 2,t 2,e1 0.0,e2 0.0,e3 0.0,e4 0.0,e5 0.0,e6 0.0}
DECL FDAT FP348={TOOL_NO 1,BASE_NO 0,IPO_FRAME #BASE}
DECL PDAT PPDAT262={VEL 100.0,ACC 100.0,APO_DIST 100.0}
DECL E6POS XP349={x 1584.68396,y -545.72821,z 1002.88202,a -35.0894089,b 3.92959905,c 179.299698,s 2,t 10,e1 0.0,e2 0.0,e3 0.0,e4 0.0,e5 0.0,e6 0.0}
DECL FDAT FP349={TOOL_NO 1,BASE_NO 0,IPO_FRAME #BASE}
DECL PDAT PPDAT263={VEL 100.0,ACC 100.0,APO_DIST 100.0}
